{region 'Components'}
// Pumps/Engines 
  fbLowPressurePump:                              FB_PUMP_WITH_BYPASS( itfOpMode:= PrgOrg.fbOpMode, 
                                                                       itfEventLogger:= PrgOrg.fbEventLogger,
                                                                       itfOn:= fbEngine_LowPressurePump_Start,
                                                                       itfBypassValve:= fbValve_LowPressureCircuit_Enable);
  fbOilCooler:                                    FB_PUMP(itfOpMode:= PrgOrg.fbOpMode,  
                                                          itfEventLogger:= PrgOrg.fbEventLogger,
                                                          itfOn:= fbEngine_OilCooler_Start);
  fbBypassPump:                                   FB_PUMP(itfOpMode:= PrgOrg.fbOpMode, 
                                                          itfEventLogger:= PrgOrg.fbEventLogger,
                                                          itfOn:= fbEngine_BypassPump_Start);
  fbCounterCyl1Pump:                              FB_PUMP_WITH_BYPASS( itfOpMode:= PrgOrg.fbOpMode, 
                                                                       itfEventLogger:= PrgOrg.fbEventLogger,
                                                                       itfOn:= fbEngine_CounterCyl1Pump_Start,
                                                                       itfBypassValve:= fbValve_CounterCyl1_Bypass);
  fbCounterCyl2Pump:                              FB_PUMP_WITH_BYPASS( itfOpMode:= PrgOrg.fbOpMode, 
                                                                       itfEventLogger:= PrgOrg.fbEventLogger,
                                                                       itfOn:= fbEngine_CounterCyl2Pump_Start,
                                                                       itfBypassValve:= fbValve_CounterCyl2_Bypass);
  fbCounterCyl3Pump:                              FB_PUMP_WITH_BYPASS( itfOpMode:= PrgOrg.fbOpMode, 
                                                                       itfEventLogger:= PrgOrg.fbEventLogger,
                                                                       itfOn:= fbEngine_CounterCyl3Pump_Start,
                                                                       itfBypassValve:= fbValve_CounterCyl3_Bypass);
  fbCounterCyl4Pump:                              FB_PUMP_WITH_BYPASS( itfOpMode:= PrgOrg.fbOpMode,  
                                                                       itfEventLogger:= PrgOrg.fbEventLogger,
                                                                       itfOn:= fbEngine_CounterCyl4Pump_Start,
                                                                       itfBypassValve:= fbValve_CounterCyl4_Bypass);
  fbTestCyl1Pump:                                 FB_PUMP(itfOpMode:= PrgOrg.fbOpMode, 
                                                          itfEventLogger:= PrgOrg.fbEventLogger,
                                                          itfOn:= fbEngine_TestCyl1Pump_Start);
  fbTestCyl2Pump:                                 FB_PUMP(itfOpMode:= PrgOrg.fbOpMode, 
                                                          itfEventLogger:= PrgOrg.fbEventLogger,
                                                          itfOn:= fbEngine_TestCyl2Pump_Start);
  fbTestCyl3Pump:                                 FB_PUMP(itfOpMode:= PrgOrg.fbOpMode, 
                                                          itfEventLogger:= PrgOrg.fbEventLogger, 
                                                          itfOn:= fbEngine_TestCyl3Pump_Start);
  fbTestCyl4Pump:                                 FB_PUMP(itfOpMode:= PrgOrg.fbOpMode, 
                                                          itfEventLogger:= PrgOrg.fbEventLogger, 
                                                          itfOn:= fbEngine_TestCyl4Pump_Start);
      
// Valves
  fbShutOffValve_LowPressure:                     FB_SHUTOFF_VALVE( itfOpMode:= PrgOrg.fbOpMode,  
                                                                    itfEventLogger:= PrgOrg.fbEventLogger,
	                                                                  itfOpen:= fbShutOffValve_Open, 
	                                                                  itfClose:= fbShutOffValve_Close,
                                                                    itfSensorOpened:= fbShutOffValve_Opened,
                                                                    itfSensorClosed:= fbShutOffValve_Closed,
                                                                    bNC:= TRUE);
  fbValve_LowPressureCircuit_Enable:              FB_VALVE_X_2( itfOpMode:= PrgOrg.fbOpMode, 
                                                                itfEventLogger:= PrgOrg.fbEventLogger,
	                                                              itfSwitchToWP:= fbValve42_LowPressureCircuit_Enable);
  fbValve_CounterCyl1_LowPressureCircuit_Add:     FB_VALVE_X_2( itfOpMode:= PrgOrg.fbOpMode, 
                                                                itfEventLogger:= PrgOrg.fbEventLogger,
	                                                              itfSwitchToWP:= fbValve42_CounterCyl1_LowPressureCircuit_Add);
  fbValve_CounterCyl2_LowPressureCircuit_Add:     FB_VALVE_X_2( itfOpMode:= PrgOrg.fbOpMode, 
                                                                itfEventLogger:= PrgOrg.fbEventLogger,
	                                                              itfSwitchToWP:= fbValve42_CounterCyl2_LowPressureCircuit_Add);
  fbValve_CounterCyl3_LowPressureCircuit_Add:     FB_VALVE_X_2( itfOpMode:= PrgOrg.fbOpMode, 
                                                                itfEventLogger:= PrgOrg.fbEventLogger,
	                                                              itfSwitchToWP:= fbValve42_CounterCyl3_LowPressureCircuit_Add);
  fbValve_CounterCyl4_LowPressureCircuit_Add:     FB_VALVE_X_2( itfOpMode:= PrgOrg.fbOpMode,  
                                                                itfEventLogger:= PrgOrg.fbEventLogger,
	                                                              itfSwitchToWP:= fbValve42_CounterCyl4_LowPressureCircuit_Add);
  fbValve_CounterCyl1:                            FB_VALVE_X_3( itfOpMode:= PrgOrg.fbOpMode, 
                                                                itfEventLogger:= PrgOrg.fbEventLogger,
	                                                              itfSwitchToWP1:= fbValve43_CounterCyl1_Extend, 
	                                                              itfSwitchToWP2:= fbValve43_CounterCyl1_Retract);
  fbValve_CounterCyl2:                            FB_VALVE_X_3( itfOpMode:= PrgOrg.fbOpMode, 
                                                                itfEventLogger:= PrgOrg.fbEventLogger,
	                                                              itfSwitchToWP1:= fbValve43_CounterCyl2_Extend, 
	                                                              itfSwitchToWP2:= fbValve43_CounterCyl2_Retract);
  fbValve_CounterCyl3:                            FB_VALVE_X_3( itfOpMode:= PrgOrg.fbOpMode, 
                                                                itfEventLogger:= PrgOrg.fbEventLogger,
	                                                              itfSwitchToWP1:= fbValve43_CounterCyl3_Extend, 
	                                                              itfSwitchToWP2:= fbValve43_CounterCyl3_Retract);
  fbValve_CounterCyl4:                            FB_VALVE_X_3( itfOpMode:= PrgOrg.fbOpMode, 
                                                                itfEventLogger:= PrgOrg.fbEventLogger,
	                                                              itfSwitchToWP1:= fbValve43_CounterCyl4_Extend, 
	                                                              itfSwitchToWP2:= fbValve43_CounterCyl4_Retract);
  fbValve_CounterCyl1JogAutoMode:                 FB_VALVE_X_2( itfOpMode:= PrgOrg.fbOpMode, 
                                                                itfEventLogger:= PrgOrg.fbEventLogger,
	                                                              itfSwitchToWP:= fbValve22_CounterCyl1_JogMode_Off);
  fbValve_CounterCyl2JogAutoMode:                 FB_VALVE_X_2( itfOpMode:= PrgOrg.fbOpMode, 
                                                                itfEventLogger:= PrgOrg.fbEventLogger,
	                                                              itfSwitchToWP:= fbValve22_CounterCyl2_JogMode_Off);
  fbValve_CounterCyl3JogAutoMode:                 FB_VALVE_X_2( itfOpMode:= PrgOrg.fbOpMode, 
                                                                itfEventLogger:= PrgOrg.fbEventLogger,
	                                                              itfSwitchToWP:= fbValve22_CounterCyl3_JogMode_Off);
  fbValve_CounterCyl4JogAutoMode:                 FB_VALVE_X_2( itfOpMode:= PrgOrg.fbOpMode,  
                                                                itfEventLogger:= PrgOrg.fbEventLogger,
	                                                              itfSwitchToWP:= fbValve22_CounterCyl4_JogMode_Off);
  fbValve_CounterCyl1_SinkBlock:                  FB_VALVE_X_2( itfOpMode:= PrgOrg.fbOpMode,  
                                                                itfEventLogger:= PrgOrg.fbEventLogger,
	                                                              itfSwitchToWP:= fbValve22_CounterCyl1_SinkBlock_Open);
  fbValve_CounterCyl2_SinkBlock:                  FB_VALVE_X_2( itfOpMode:= PrgOrg.fbOpMode,  
                                                                itfEventLogger:= PrgOrg.fbEventLogger,
	                                                              itfSwitchToWP:= fbValve22_CounterCyl2_SinkBlock_Open);
  fbValve_CounterCyl3_SinkBlock:                  FB_VALVE_X_2( itfOpMode:= PrgOrg.fbOpMode,  
                                                                itfEventLogger:= PrgOrg.fbEventLogger,
	                                                              itfSwitchToWP:= fbValve22_CounterCyl3_SinkBlock_Open);
  fbValve_CounterCyl4_SinkBlock:                  FB_VALVE_X_2( itfOpMode:= PrgOrg.fbOpMode,  
                                                                itfEventLogger:= PrgOrg.fbEventLogger,
	                                                              itfSwitchToWP:= fbValve22_CounterCyl4_SinkBlock_Open);
  fbValve_CounterCyl1_WorkPressure:               FB_PRV_PROP(itfOpMode:= PrgOrg.fbOpMode, 
                                                              itfEventLogger:= PrgOrg.fbEventLogger,
                                                              rMaxLimitInBar:= 275.0);
  fbValve_CounterCyl2_WorkPressure:               FB_PRV_PROP(itfOpMode:= PrgOrg.fbOpMode, 
                                                              itfEventLogger:= PrgOrg.fbEventLogger,
                                                              rMaxLimitInBar:= 275.0);
  fbValve_CounterCyl3_WorkPressure:               FB_PRV_PROP(itfOpMode:= PrgOrg.fbOpMode, 
                                                              itfEventLogger:= PrgOrg.fbEventLogger,
                                                              rMaxLimitInBar:= 275.0);
  fbValve_CounterCyl4_WorkPressure:               FB_PRV_PROP(itfOpMode:= PrgOrg.fbOpMode, 
                                                              itfEventLogger:= PrgOrg.fbEventLogger,
                                                              rMaxLimitInBar:= 275.0);
  fbValve_CounterCyl1_Bypass:                     FB_VALVE_X_2( itfOpMode:= PrgOrg.fbOpMode, 
                                                                itfEventLogger:= PrgOrg.fbEventLogger,
	                                                              itfSwitchToWP:= fbValve42_CounterCyl1_Bypass_Add);
  fbValve_CounterCyl2_Bypass:                     FB_VALVE_X_2( itfOpMode:= PrgOrg.fbOpMode, 
                                                                itfEventLogger:= PrgOrg.fbEventLogger, 
	                                                              itfSwitchToWP:= fbValve42_CounterCyl2_Bypass_Add);
  fbValve_CounterCyl3_Bypass:                     FB_VALVE_X_2( itfOpMode:= PrgOrg.fbOpMode,  
                                                                itfEventLogger:= PrgOrg.fbEventLogger,
	                                                              itfSwitchToWP:= fbValve42_CounterCyl3_Bypass_Add);
  fbValve_CounterCyl4_Bypass:                     FB_VALVE_X_2( itfOpMode:= PrgOrg.fbOpMode, 
                                                                itfEventLogger:= PrgOrg.fbEventLogger,
	                                                              itfSwitchToWP:= fbValve42_CounterCyl4_Bypass_Add);
  fbValve_TestCyl1:                               FB_VALVE_X_3_PROP(itfOpMode:= PrgOrg.fbOpMode, 
                                                                    itfEventLogger:= PrgOrg.fbEventLogger);
  fbValve_TestCyl2:                               FB_VALVE_X_3_PROP(itfOpMode:= PrgOrg.fbOpMode, 
                                                                    itfEventLogger:= PrgOrg.fbEventLogger);
  fbValve_TestCyl3:                               FB_VALVE_X_3_PROP(itfOpMode:= PrgOrg.fbOpMode, 
                                                                    itfEventLogger:= PrgOrg.fbEventLogger);
  fbValve_TestCyl4:                               FB_VALVE_X_3_PROP(itfOpMode:= PrgOrg.fbOpMode, 
                                                                    itfEventLogger:= PrgOrg.fbEventLogger);
  fbValve_TestCyl1_A_Unlock:                      FB_VALVE_X_2( itfOpMode:= PrgOrg.fbOpMode, 
                                                                itfEventLogger:= PrgOrg.fbEventLogger,
	                                                              itfSwitchToWP:= fbValve22_TestCyl1_A_Open);
  fbValve_TestCyl1_B_Unlock:                      FB_VALVE_X_2( itfOpMode:= PrgOrg.fbOpMode, 
                                                                itfEventLogger:= PrgOrg.fbEventLogger, 
	                                                              itfSwitchToWP:= fbValve22_TestCyl1_B_Open);
  fbValve_TestCyl2_A_Unlock:                      FB_VALVE_X_2( itfOpMode:= PrgOrg.fbOpMode,   
                                                                itfEventLogger:= PrgOrg.fbEventLogger, 
	                                                              itfSwitchToWP:= fbValve22_TestCyl2_A_Open);
  fbValve_TestCyl2_B_Unlock:                      FB_VALVE_X_2( itfOpMode:= PrgOrg.fbOpMode, 
                                                                itfEventLogger:= PrgOrg.fbEventLogger,  
	                                                              itfSwitchToWP:= fbValve22_TestCyl2_B_Open);
  fbValve_TestCyl3_A_Unlock:                      FB_VALVE_X_2( itfOpMode:= PrgOrg.fbOpMode,  
                                                                itfEventLogger:= PrgOrg.fbEventLogger,
	                                                              itfSwitchToWP:= fbValve22_TestCyl3_A_Open);
  fbValve_TestCyl3_B_Unlock:                      FB_VALVE_X_2( itfOpMode:= PrgOrg.fbOpMode,  
                                                                itfEventLogger:= PrgOrg.fbEventLogger,
	                                                              itfSwitchToWP:= fbValve22_TestCyl3_B_Open);
  fbValve_TestCyl4_A_Unlock:                      FB_VALVE_X_2( itfOpMode:= PrgOrg.fbOpMode, 
                                                                itfEventLogger:= PrgOrg.fbEventLogger,
	                                                              itfSwitchToWP:= fbValve22_TestCyl4_A_Open);
  fbValve_TestCyl4_B_Unlock:                      FB_VALVE_X_2( itfOpMode:= PrgOrg.fbOpMode, 
                                                                itfEventLogger:= PrgOrg.fbEventLogger,
	                                                              itfSwitchToWP:= fbValve22_TestCyl4_B_Open);
  fbValve_TestCyl1_WorkPressure:                  FB_PRV_PROP(itfOpMode:= PrgOrg.fbOpMode, 
                                                              itfEventLogger:= PrgOrg.fbEventLogger,
                                                              rMaxLimitInBar:= 275.0);
  fbValve_TestCyl2_WorkPressure:                  FB_PRV_PROP(itfOpMode:= PrgOrg.fbOpMode, 
                                                              itfEventLogger:= PrgOrg.fbEventLogger,
                                                              rMaxLimitInBar:= 275.0);
  fbValve_TestCyl3_WorkPressure:                  FB_PRV_PROP(itfOpMode:= PrgOrg.fbOpMode, 
                                                              itfEventLogger:= PrgOrg.fbEventLogger,
                                                              rMaxLimitInBar:= 275.0);
  fbValve_TestCyl4_WorkPressure:                  FB_PRV_PROP(itfOpMode:= PrgOrg.fbOpMode, 
                                                              itfEventLogger:= PrgOrg.fbEventLogger,
                                                              rMaxLimitInBar:= 275.0);
  fbValve_TestCyl1_LowPressure:                   FB_PRV_PROP(itfOpMode:= PrgOrg.fbOpMode, 
                                                              itfEventLogger:= PrgOrg.fbEventLogger,
                                                              rMaxLimitInBar:= 25.0);
  fbValve_Pump4_Add:                              FB_VALVE_X_2( itfOpMode:= PrgOrg.fbOpMode, 
                                                                itfEventLogger:= PrgOrg.fbEventLogger,
	                                                              itfSwitchToWP:= fbValve22_Pump4_Add);
  fbValve_Pump3_Add:                              FB_VALVE_X_2( itfOpMode:= PrgOrg.fbOpMode,  
                                                                itfEventLogger:= PrgOrg.fbEventLogger,
	                                                              itfSwitchToWP:= fbValve22_Pump3_Add);
  fbValve_Pump2_Add:                              FB_VALVE_X_2( itfOpMode:= PrgOrg.fbOpMode,  
                                                                itfEventLogger:= PrgOrg.fbEventLogger,
	                                                              itfSwitchToWP:= fbValve22_Pump2_Add);
  fbValve_PressureReservoir_A_Add:                FB_VALVE_X_2( itfOpMode:= PrgOrg.fbOpMode, 
                                                                itfEventLogger:= PrgOrg.fbEventLogger, 
	                                                              itfSwitchToWP:= fbValve22_PressureReservoir_A_Add);
  fbValve_PressureReservoir_B_Add:                FB_VALVE_X_2( itfOpMode:= PrgOrg.fbOpMode, 
                                                                itfEventLogger:= PrgOrg.fbEventLogger,
	                                                              itfSwitchToWP:= fbValve22_PressureReservoir_B_Add);
  fbValve_SensorBreakPressure_A_Add:              FB_VALVE_X_2( itfOpMode:= PrgOrg.fbOpMode, 
                                                                itfEventLogger:= PrgOrg.fbEventLogger,
	                                                              itfSwitchToWP:= fbValve32_SensorBreakPressure_A_Add);
  fbValve_SensorBreakPressure_B_Add:              FB_VALVE_X_2( itfOpMode:= PrgOrg.fbOpMode, 
                                                                itfEventLogger:= PrgOrg.fbEventLogger,
	                                                              itfSwitchToWP:= fbValve32_SensorBreakPressure_B_Add);
                                                  
// Cylinders                                      
  fbCounterCyl1:                                  FB_CYLINDER_DA_COUNTER( itfOpMode:= PrgOrg.fbOpMode, 
                                                                          itfEventLogger:= PrgOrg.fbEventLogger,
                                                                          itfOpModeVisu:= PrgVisu.fbVisuOPMode,
                                                                          itfValve_CylCtrl:= fbValve_CounterCyl1,
                                                                          itfValve_Bypass:= fbValve_CounterCyl1_Bypass,
                                                                          itfValve_AutomaticEnable:= fbValve_CounterCyl1JogAutoMode,
                                                                          itfValve_SinkBlock:= fbValve_CounterCyl1_SinkBlock,
                                                                          itfValve_LowPressureCircuitAdd:= fbValve_CounterCyl1_LowPressureCircuit_Add,
                                                                          itfValve_PressureLimit:= fbValve_CounterCyl1_WorkPressure,
                                                                          itfJogBtnPos_Pressed:= fbJogBtnPos_Pressed,
                                                                          itfJogBtnNeg_Pressed:= fbJogBtnNeg_Pressed,
	                                                                        lrPistonSurfaceA:= 1963.495, 
	                                                                        lrPistonSurfaceB:= 962.112, 
	                                                                        rEndPosTol:= 1,
                                                                          rPumpVolumeFlow:= 4.0,
                                                                          rPumpEfficiencyFactor:= 0.85);
  fbCounterCyl2:                                  FB_CYLINDER_DA_COUNTER( itfOpMode:= PrgOrg.fbOpMode, 
                                                                          itfEventLogger:= PrgOrg.fbEventLogger,
                                                                          itfOpModeVisu:= PrgVisu.fbVisuOPMode,
                                                                          itfValve_CylCtrl:= fbValve_CounterCyl2,
                                                                          itfValve_Bypass:= fbValve_CounterCyl2_Bypass,
                                                                          itfValve_AutomaticEnable:= fbValve_CounterCyl2JogAutoMode,
                                                                          itfValve_SinkBlock:= fbValve_CounterCyl2_SinkBlock,
                                                                          itfValve_LowPressureCircuitAdd:= fbValve_CounterCyl2_LowPressureCircuit_Add,
                                                                          itfValve_PressureLimit:= fbValve_CounterCyl2_WorkPressure,
                                                                          itfJogBtnPos_Pressed:= fbJogBtnPos_Pressed,
                                                                          itfJogBtnNeg_Pressed:= fbJogBtnNeg_Pressed,
	                                                                        lrPistonSurfaceA:= 1963.495, 
	                                                                        lrPistonSurfaceB:= 962.112, 
	                                                                        rEndPosTol:= 1,
                                                                          rPumpVolumeFlow:= 4.0,
                                                                          rPumpEfficiencyFactor:= 0.85);
  fbCounterCyl3:                                  FB_CYLINDER_DA_COUNTER( itfOpMode:= PrgOrg.fbOpMode, 
                                                                          itfEventLogger:= PrgOrg.fbEventLogger,
                                                                          itfOpModeVisu:= PrgVisu.fbVisuOPMode,
                                                                          itfValve_CylCtrl:= fbValve_CounterCyl3,
                                                                          itfValve_Bypass:= fbValve_CounterCyl3_Bypass,
                                                                          itfValve_AutomaticEnable:= fbValve_CounterCyl3JogAutoMode,
                                                                          itfValve_SinkBlock:= fbValve_CounterCyl3_SinkBlock,
                                                                          itfValve_LowPressureCircuitAdd:= fbValve_CounterCyl3_LowPressureCircuit_Add,
                                                                          itfValve_PressureLimit:= fbValve_CounterCyl3_WorkPressure,
                                                                          itfJogBtnPos_Pressed:= fbJogBtnPos_Pressed,
                                                                          itfJogBtnNeg_Pressed:= fbJogBtnNeg_Pressed,
	                                                                        lrPistonSurfaceA:= 1963.495, 
	                                                                        lrPistonSurfaceB:= 962.112, 
	                                                                        rEndPosTol:= 1,
                                                                          rPumpVolumeFlow:= 4.0,
                                                                          rPumpEfficiencyFactor:= 0.85);
  fbCounterCyl4:                                  FB_CYLINDER_DA_COUNTER( itfOpMode:= PrgOrg.fbOpMode, 
                                                                          itfEventLogger:= PrgOrg.fbEventLogger,
                                                                          itfOpModeVisu:= PrgVisu.fbVisuOPMode,
                                                                          itfValve_CylCtrl:= fbValve_CounterCyl4,
                                                                          itfValve_Bypass:= fbValve_CounterCyl4_Bypass,
                                                                          itfValve_AutomaticEnable:= fbValve_CounterCyl4JogAutoMode,
                                                                          itfValve_SinkBlock:= fbValve_CounterCyl4_SinkBlock,
                                                                          itfValve_LowPressureCircuitAdd:= fbValve_CounterCyl4_LowPressureCircuit_Add,
                                                                          itfValve_PressureLimit:= fbValve_CounterCyl4_WorkPressure,  
                                                                          itfJogBtnPos_Pressed:= fbJogBtnPos_Pressed,
                                                                          itfJogBtnNeg_Pressed:= fbJogBtnNeg_Pressed,
	                                                                        lrPistonSurfaceA:= 1963.495, 
	                                                                        lrPistonSurfaceB:= 962.112, 
	                                                                        rEndPosTol:= 1,
                                                                          rPumpVolumeFlow:= 4.0,
                                                                          rPumpEfficiencyFactor:= 0.85);
  fbTestCyl1:                                     FB_CYLINDER_DA_TESTDEV1(itfOpMode:= PrgOrg.fbOpMode, 
                                                                          itfEventLogger:= PrgOrg.fbEventLogger, 
                                                                          itfOpModeVisu:= PrgVisu.fbVisuOPMode,
	                                                                        itfValve_CylCtrl:= fbValve_TestCyl1, 
	                                                                        itfValve_LockA:= fbValve_TestCyl1_A_Unlock, 
	                                                                        itfValve_LockB:= fbValve_TestCyl1_B_Unlock, 
	                                                                        itfValve_AddPump2:= fbValve_Pump2_Add, 
	                                                                        itfValve_AddPump3:= fbValve_Pump3_Add, 
	                                                                        itfValve_AddPump4:= fbValve_Pump4_Add, 
	                                                                        itfValve_PressureReservoirAAdd:= fbValve_PressureReservoir_A_Add, 
	                                                                        itfValve_PressureReservoirBAdd:= fbValve_PressureReservoir_B_Add, 
	                                                                        itfValve_SensorBreakPressureAAdd:= fbValve_SensorBreakPressure_A_Add, 
	                                                                        itfValve_SensorBreakPressureBAdd:= fbValve_SensorBreakPressure_B_Add, 
	                                                                        fbShutOffValve_LowPressure:= fbShutOffValve_LowPressure, 
	                                                                        itfValve_PressureLimit:= fbValve_TestCyl1_WorkPressure, 
	                                                                        itfValve_LowPressureLimit:= fbValve_TestCyl1_LowPressure,
                                                                          itfPumpMain:= fbTestCyl1Pump,
                                                                          itfPump2:= fbTestCyl2Pump, 
                                                                          itfPump3:= fbTestCyl3Pump, 
                                                                          itfPump4:= fbTestCyl4Pump, 
	                                                                        rEndPosTol:= 1,
                                                                          rPumpVolumeFlow:= 3.0,
                                                                          rPumpEfficiencyFactor:= 0.85);
  fbTestCyl2:                                     FB_CYLINDER_DA_TESTDEV2_4(itfOpMode:= PrgOrg.fbOpMode, 
                                                                            itfEventLogger:= PrgOrg.fbEventLogger,
                                                                            itfOpModeVisu:= PrgVisu.fbVisuOPMode,
	                                                                          itfValve_CylCtrl:= fbValve_TestCyl2, 
	                                                                          itfValve_LockA:= fbValve_TestCyl2_A_Unlock, 
	                                                                          itfValve_LockB:= fbValve_TestCyl2_B_Unlock, 
	                                                                          itfValve_PressureLimit:= fbValve_TestCyl2_WorkPressure,
	                                                                          rEndPosTol:= 1,
                                                                            rPumpVolumeFlow:= 3.0,
                                                                            rPumpEfficiencyFactor:= 0.85);
  fbTestCyl3:                                     FB_CYLINDER_DA_TESTDEV2_4(itfOpMode:= PrgOrg.fbOpMode,  
                                                                            itfEventLogger:= PrgOrg.fbEventLogger,
                                                                            itfOpModeVisu:= PrgVisu.fbVisuOPMode,
	                                                                          itfValve_CylCtrl:= fbValve_TestCyl3, 
	                                                                          itfValve_LockA:= fbValve_TestCyl3_A_Unlock, 
	                                                                          itfValve_LockB:= fbValve_TestCyl3_B_Unlock, 
	                                                                          itfValve_PressureLimit:= fbValve_TestCyl3_WorkPressure, 
	                                                                          rEndPosTol:= 1,
                                                                            rPumpVolumeFlow:= 3.0,
                                                                            rPumpEfficiencyFactor:= 0.85);
  fbTestCyl4:                                     FB_CYLINDER_DA_TESTDEV2_4(itfOpMode:= PrgOrg.fbOpMode, 
                                                                            itfEventLogger:= PrgOrg.fbEventLogger,
                                                                            itfOpModeVisu:= PrgVisu.fbVisuOPMode,
	                                                                          itfValve_CylCtrl:= fbValve_TestCyl4, 
	                                                                          itfValve_LockA:= fbValve_TestCyl4_A_Unlock, 
	                                                                          itfValve_LockB:= fbValve_TestCyl4_B_Unlock, 
	                                                                          itfValve_PressureLimit:= fbValve_TestCyl4_WorkPressure,
	                                                                          rEndPosTol:= 1,
                                                                            rPumpVolumeFlow:= 3.0,
                                                                            rPumpEfficiencyFactor:= 0.85);
{endregion}
   
{region 'Main process'}
  fbNest1:                                        FB_SEQ_PROCESS_NEST1( itfOpMode:= PrgOrg.fbOpMode, 
                                                                        itfEventLogger:= PrgOrg.fbEventLogger,
                                                                        itfTimer:= fbTimerNest1, 
	                                                                      itfCounterCyl:= fbCounterCyl1, 
	                                                                      itfTestCyl:= fbTestCyl1, 
	                                                                      itfCounterCylPump:= fbCounterCyl1Pump, 
	                                                                      itfTestCylPump:= fbTestCyl1Pump,
                                                                        itfPump2Pressure:= fbValve_TestCyl2_WorkPressure,
                                                                        itfPump3Pressure:= fbValve_TestCyl3_WorkPressure,
                                                                        itfPump4Pressure:= fbValve_TestCyl4_WorkPressure);
  fbNest2:                                        FB_SEQ_PROCESS_NEST2_4( itfOpMode:= PrgOrg.fbOpMode, 
                                                                          itfEventLogger:= PrgOrg.fbEventLogger,
                                                                          itfTimer:= fbTimerNest2, 
	                                                                        itfCounterCyl:= fbCounterCyl2, 
	                                                                        itfTestCyl:= fbTestCyl2, 
	                                                                        itfCounterCylPump:= fbCounterCyl2Pump, 
	                                                                        itfTestCylPump:= fbTestCyl2Pump);
  fbNest3:                                        FB_SEQ_PROCESS_NEST2_4( itfOpMode:= PrgOrg.fbOpMode,  
                                                                          itfEventLogger:= PrgOrg.fbEventLogger,
                                                                          itfTimer:= fbTimerNest3,
	                                                                        itfCounterCyl:= fbCounterCyl3, 
	                                                                        itfTestCyl:= fbTestCyl3, 
	                                                                        itfCounterCylPump:= fbCounterCyl3Pump, 
	                                                                        itfTestCylPump:= fbTestCyl3Pump);
  fbNest4:                                        FB_SEQ_PROCESS_NEST2_4( itfOpMode:= PrgOrg.fbOpMode,  
                                                                          itfEventLogger:= PrgOrg.fbEventLogger,
                                                                          itfTimer:= fbTimerNest4,
	                                                                        itfCounterCyl:= fbCounterCyl4, 
	                                                                        itfTestCyl:= fbTestCyl4, 
	                                                                        itfCounterCylPump:= fbCounterCyl4Pump, 
	                                                                        itfTestCylPump:= fbTestCyl4Pump);
  fbMainProcess:                                  FB_PROCESS_MAIN(itfOpMode:= PrgOrg.fbOpMode, 
                                                                  itfEventLogger:= PrgOrg.fbEventLogger, 
                                                                  itfTimerNest1:= fbTimerNest1,
                                                                  itfTimerNest2:= fbTimerNest2,
                                                                  itfTimerNest3:= fbTimerNest3,
                                                                  itfTimerNest4:= fbTimerNest4,
	                                                                itfNest1:= fbNest1, 
	                                                                itfNest2:= fbNest2, 
	                                                                itfNest3:= fbNest3, 
	                                                                itfNest4:= fbNest4, 
	                                                                itfLowPressurePump:= fbLowPressurePump, 
	                                                                itfOilCooler:= fbOilCooler, 
	                                                                itfBypassPump:= fbBypassPump,
                                                                  itfLevelSwitch_AggregateTank1_Out1:= fbLevelSwitch_AggregateTank1_Out1,
                                                                  itfLevelSwitch_AggregateTank1_Out2:= fbLevelSwitch_AggregateTank1_Out2,
                                                                  itfTemperatureSwitch_AggregateTank1_Out1:= fbTemperatureSwitch_AggregateTank1_Out1,
                                                                  itfTemperatureSwitch_AggregateTank1_Out2:= fbTemperatureSwitch_AggregateTank1_Out2,
                                                                  itfLevelSwitch_AggregateTank2_Out1:= fbLevelSwitch_AggregateTank2_Out1,
                                                                  itfLevelSwitch_AggregateTank2_Out2:= fbLevelSwitch_AggregateTank2_Out2,
                                                                  itfLevelSwitch_AggregateTank2_Out3:= fbLevelSwitch_AggregateTank2_Out3,
                                                                  itfSwitch_AggregateFilter_Dirty:= fbSwitch_AggregateFilter_Dirty);
{endregion}
   
{region 'Recipe'}
  stRecipeParams:                                 ST_RECIPE_PARAMS;
{endregion}
END_VAR
VAR
  rMaxSpeedInMmPerSHP:                            REAL;
  rMaxSpeedInMmPerSWP:                            REAL;
END_VAR

VAR PERSISTENT
  stSettings:                                     ST_SETTINGS;
  sTestCyl1SNo:                                   STRING := '';
  sTestCyl2SNo:                                   STRING := '';
  sTestCyl3SNo:                                   STRING := '';
  sTestCyl4SNo:                                   STRING := '';
END_VAR

(* Actions *)
A_000_FBs();
A_010_InputToBNC();
A_020_SetObjectPath();
A_030_OilCooler();
A_040_MachineLight();
A_100_Control();

ACTION A_000_FBs:
(* FBs *)
// General
fbTimerNest1();
fbTimerNest2();
fbTimerNest3();
fbTimerNest4();
rPressureConverted_TestCyl1 := TO_REAL(iPressureSensor_TestCyl1) * 0.025;
rPressureConverted_TestCyl1_A := TO_REAL(iPressureSensor_TestCyl1_A) * 0.025;
rPressureConverted_TestCyl1_B := TO_REAL(iPressureSensor_TestCyl1_B) * 0.025;
rPressureConverted_CounterCyl1 := TO_REAL(iPressureSensor_CounterCyl1) * 0.025;
rPressureConverted_LowPressure := TO_REAL(iPressureSensor_LowPressure) * 0.001;
rPressureConverted_TestCyl1_BreakPressure_A := TO_REAL(iPressureSensor_TestCyl1_BreakPressure_A) * 0.001;
rPressureConverted_TestCyl1_BreakPressure_B := TO_REAL(iPressureSensor_TestCyl1_BreakPressure_B) * 0.001;
rPressureConverted_TestCyl1_PressureReservoir := TO_REAL(iPressureSensor_TestCyl1_PressureReservoir) * 0.025;
rPressureConverted_TestCyl2 := TO_REAL(iPressureSensor_TestCyl2) * 0.025;
rPressureConverted_TestCyl2_A := TO_REAL(iPressureSensor_TestCyl2_A) * 0.025;
rPressureConverted_TestCyl2_B := TO_REAL(iPressureSensor_TestCyl2_B) * 0.025;
rPressureConverted_CounterCyl2 := TO_REAL(iPressureSensor_CounterCyl2) * 0.025;
rPressureConverted_TestCyl3 := TO_REAL(iPressureSensor_TestCyl3) * 0.025;
rPressureConverted_TestCyl3_A := TO_REAL(iPressureSensor_TestCyl3_A) * 0.025;
rPressureConverted_TestCyl3_B := TO_REAL(iPressureSensor_TestCyl3_B) * 0.025;
rPressureConverted_CounterCyl3 := TO_REAL(iPressureSensor_CounterCyl3) * 0.025;
rPressureConverted_TestCyl4 := TO_REAL(iPressureSensor_TestCyl4) * 0.025;
rPressureConverted_TestCyl4_A := TO_REAL(iPressureSensor_TestCyl4_A) * 0.025;
rPressureConverted_TestCyl4_B := TO_REAL(iPressureSensor_TestCyl4_B) * 0.025;
rPressureConverted_CounterCyl4 := TO_REAL(iPressureSensor_CounterCyl4) * 0.025;


// Pmps/Engines
fbLowPressurePump();
fbOilCooler();
fbBypassPump();
fbCounterCyl1Pump();
fbCounterCyl2Pump();
fbCounterCyl3Pump();
fbCounterCyl4Pump();
fbTestCyl1Pump();
fbTestCyl2Pump();
fbTestCyl3Pump();
fbTestCyl4Pump();
fbShutOffValve_LowPressure();

// Valves
fbValve_LowPressureCircuit_Enable();
fbValve_CounterCyl1_LowPressureCircuit_Add();
fbValve_CounterCyl2_LowPressureCircuit_Add();
fbValve_CounterCyl3_LowPressureCircuit_Add();
fbValve_CounterCyl4_LowPressureCircuit_Add();
fbValve_CounterCyl1();
fbValve_CounterCyl2();
fbValve_CounterCyl3();
fbValve_CounterCyl4();
fbValve_CounterCyl1JogAutoMode();
fbValve_CounterCyl2JogAutoMode();
fbValve_CounterCyl3JogAutoMode();
fbValve_CounterCyl4JogAutoMode();
fbValve_CounterCyl1_SinkBlock();
fbValve_CounterCyl2_SinkBlock();
fbValve_CounterCyl3_SinkBlock();
fbValve_CounterCyl4_SinkBlock();
fbValve_CounterCyl1_WorkPressure(iTargetVal=> iCounterCyl1_Pressure);
fbValve_CounterCyl2_WorkPressure(iTargetVal=> iCounterCyl2_Pressure);
fbValve_CounterCyl3_WorkPressure(iTargetVal=> iCounterCyl3_Pressure);
fbValve_CounterCyl4_WorkPressure(iTargetVal=> iCounterCyl4_Pressure);
fbValve_CounterCyl1_Bypass();
fbValve_CounterCyl2_Bypass();
fbValve_CounterCyl3_Bypass();
fbValve_CounterCyl4_Bypass();
fbValve_TestCyl1(iAnalogSwitch=> iValve43_TestCyl1);
fbValve_TestCyl2(iAnalogSwitch=> iValve43_TestCyl2);
fbValve_TestCyl3(iAnalogSwitch=> iValve43_TestCyl3);
fbValve_TestCyl4(iAnalogSwitch=> iValve43_TestCyl4);
fbValve_TestCyl1_A_Unlock();
fbValve_TestCyl1_B_Unlock();
fbValve_TestCyl2_A_Unlock();
fbValve_TestCyl2_B_Unlock();
fbValve_TestCyl3_A_Unlock();
fbValve_TestCyl3_B_Unlock();
fbValve_TestCyl4_A_Unlock();
fbValve_TestCyl4_B_Unlock();
fbValve_TestCyl1_WorkPressure(iTargetVal=> iTestCyl1_Pressure);
fbValve_TestCyl2_WorkPressure(iTargetVal=> iTestCyl2_Pressure);
fbValve_TestCyl3_WorkPressure(iTargetVal=> iTestCyl3_Pressure);
fbValve_TestCyl4_WorkPressure(iTargetVal=> iTestCyl4_Pressure);
fbValve_TestCyl1_LowPressure(iTargetVal=> iTestCyl1_LowPressure);
fbValve_Pump4_Add();
fbValve_Pump3_Add();
fbValve_Pump2_Add();
fbValve_PressureReservoir_A_Add();
fbValve_PressureReservoir_B_Add();
fbValve_SensorBreakPressure_A_Add();
fbValve_SensorBreakPressure_B_Add();

// Cylinders
fbCounterCyl1(rCurrentPressureInBar:= rPressureConverted_CounterCyl1, 
              bJogActive:= PrgVisu.fbVisuOPMode.P_JogCounterCyl1_Active,
              rPressureRegulationFactor:= stSettings.rPressureRegulationFactor,
              rPressureRegulationTolerance:= stSettings.rPressureRegulationTolerance);
fbCounterCyl2(rCurrentPressureInBar:= rPressureConverted_CounterCyl2, 
              bJogActive:= PrgVisu.fbVisuOPMode.P_JogCounterCyl2_Active,
              rPressureRegulationFactor:= stSettings.rPressureRegulationFactor,
              rPressureRegulationTolerance:= stSettings.rPressureRegulationTolerance);
fbCounterCyl3(rCurrentPressureInBar:= rPressureConverted_CounterCyl3, 
              bJogActive:= PrgVisu.fbVisuOPMode.P_JogCounterCyl3_Active,
              rPressureRegulationFactor:= stSettings.rPressureRegulationFactor,
              rPressureRegulationTolerance:= stSettings.rPressureRegulationTolerance);
fbCounterCyl4(rCurrentPressureInBar:= rPressureConverted_CounterCyl4, 
              bJogActive:= PrgVisu.fbVisuOPMode.P_JogCounterCyl4_Active,
              rPressureRegulationFactor:= stSettings.rPressureRegulationFactor,
              rPressureRegulationTolerance:= stSettings.rPressureRegulationTolerance);
fbTestCyl1( bDoableActing:= stRecipeParams.stRecipeCyl.bDoubleActing,
            lrCurrentPosAbs:= TO_LREAL(diTestCyl1_Distance), 
            rCurrentPressureInBar:= rPressureConverted_TestCyl1,
            rCurrentPressureInBarA:= rPressureConverted_TestCyl1_A,
            rCurrentPressureInBarB:= rPressureConverted_TestCyl1_B,
            rCurrentLowPressureInBar:= rPressureConverted_LowPressure,
            rCurrentLowPressureInBarA:= rPressureConverted_TestCyl1_BreakPressure_A,
            rCurrentLowPressureInBarB:= rPressureConverted_TestCyl1_BreakPressure_B,
            rCurrentReservoirPressureInBar:= rPressureConverted_TestCyl1_PressureReservoir,
            lrPistonSurfaceA:= stRecipeParams.stRecipeCyl.lrPistonSurfaceA,
            lrPistonSurfaceB:= stRecipeParams.stRecipeCyl.lrPistonSurfaceB,
            rSpeedRegulationFactor:= stSettings.rSpeedRegulationFactor,
            rSpeedRegulationTolerance:= stSettings.rSpeedRegulationTolerance,
            rPressureRegulationFactor:= stSettings.rPressureRegulationFactor,
            rPressureRegulationTolerance:= stSettings.rPressureRegulationTolerance);
fbTestCyl2( bDoableActing:= stRecipeParams.stRecipeCyl.bDoubleActing,
            lrCurrentPosAbs:= TO_REAL(diTestCyl2_Distance), 
            rCurrentPressureInBar:= rPressureConverted_TestCyl2,
            rCurrentPressureInBarA:= rPressureConverted_TestCyl2_A,
            rCurrentPressureInBarB:= rPressureConverted_TestCyl2_B,
            lrPistonSurfaceA:= stRecipeParams.stRecipeCyl.lrPistonSurfaceA,
            lrPistonSurfaceB:= stRecipeParams.stRecipeCyl.lrPistonSurfaceB,
            rSpeedRegulationFactor:= stSettings.rSpeedRegulationFactor,
            rSpeedRegulationTolerance:= stSettings.rSpeedRegulationTolerance,
            rPressureRegulationFactor:= stSettings.rPressureRegulationFactor,
            rPressureRegulationTolerance:= stSettings.rPressureRegulationTolerance);
fbTestCyl3( bDoableActing:= stRecipeParams.stRecipeCyl.bDoubleActing,
            lrCurrentPosAbs:= TO_REAL(diTestCyl3_Distance), 
            rCurrentPressureInBar:= rPressureConverted_TestCyl3,
            rCurrentPressureInBarA:= rPressureConverted_TestCyl3_A,
            rCurrentPressureInBarB:= rPressureConverted_TestCyl3_B,
            lrPistonSurfaceA:= stRecipeParams.stRecipeCyl.lrPistonSurfaceA,
            lrPistonSurfaceB:= stRecipeParams.stRecipeCyl.lrPistonSurfaceB,
            rSpeedRegulationFactor:= stSettings.rSpeedRegulationFactor,
            rSpeedRegulationTolerance:= stSettings.rSpeedRegulationTolerance,
            rPressureRegulationFactor:= stSettings.rPressureRegulationFactor,
            rPressureRegulationTolerance:= stSettings.rPressureRegulationTolerance);
fbTestCyl4( bDoableActing:= stRecipeParams.stRecipeCyl.bDoubleActing,
            lrCurrentPosAbs:= TO_REAL(diTestCyl4_Distance), 
            rCurrentPressureInBar:= rPressureConverted_TestCyl4,
            rCurrentPressureInBarA:= rPressureConverted_TestCyl4_A,
            rCurrentPressureInBarB:= rPressureConverted_TestCyl4_B,
            lrPistonSurfaceA:= stRecipeParams.stRecipeCyl.lrPistonSurfaceA,
            lrPistonSurfaceB:= stRecipeParams.stRecipeCyl.lrPistonSurfaceB,
            rSpeedRegulationFactor:= stSettings.rSpeedRegulationFactor,
            rSpeedRegulationTolerance:= stSettings.rSpeedRegulationTolerance,
            rPressureRegulationFactor:= stSettings.rPressureRegulationFactor,
            rPressureRegulationTolerance:= stSettings.rPressureRegulationTolerance);

// Main process
fbNest1(bDoubleActing:= stRecipeParams.stRecipeCyl.bDoubleActing,
        rMaxSpeedInMmPerSHP=> rMaxSpeedInMmPerSHP,
        rMaxSpeedInMmPerSWP=> rMaxSpeedInMmPerSWP,
        rSpeedEfficiencyFactor:= stSettings.rSpeedEfficiencyFactor,
        uiRecordDelay:= stSettings.uiRecordDelay);
fbNest2(bDoubleActing:= stRecipeParams.stRecipeCyl.bDoubleActing,
        rMaxSpeedInMmPerSHP:= rMaxSpeedInMmPerSHP,
        rMaxSpeedInMmPerSWP:= rMaxSpeedInMmPerSWP,
        rSpeedEfficiencyFactor:= stSettings.rSpeedEfficiencyFactor,
        uiRecordDelay:= stSettings.uiRecordDelay);
fbNest3(bDoubleActing:= stRecipeParams.stRecipeCyl.bDoubleActing,
        rMaxSpeedInMmPerSHP:= rMaxSpeedInMmPerSHP,
        rMaxSpeedInMmPerSWP:= rMaxSpeedInMmPerSWP,
        rSpeedEfficiencyFactor:= stSettings.rSpeedEfficiencyFactor,
        uiRecordDelay:= stSettings.uiRecordDelay);
fbNest4(bDoubleActing:= stRecipeParams.stRecipeCyl.bDoubleActing,
        rMaxSpeedInMmPerSHP:= rMaxSpeedInMmPerSHP,
        rMaxSpeedInMmPerSWP:= rMaxSpeedInMmPerSWP,
        rSpeedEfficiencyFactor:= stSettings.rSpeedEfficiencyFactor,
        uiRecordDelay:= stSettings.uiRecordDelay);
fbMainProcess();
END_ACTION

ACTION A_010_InputToBNC:
iBNCSocket_TestCyl1_A_Pressure := TO_INT(rPressureConverted_TestCyl1_A);
iBNCSocket_TestCyl1_B_Pressure := TO_INT(rPressureConverted_TestCyl1_B);
iBNCSocket_CounterCyl1_Pressure := TO_INT(rPressureConverted_CounterCyl1);
iBNCSocket_TestCyl1_Distance := TO_INT(diTestCyl1_Distance);
iBNCSocket_TestCyl1_A_BreakPressure := iPressureSensor_TestCyl1_BreakPressure_A;
iBNCSocket_TestCyl1_B_BreakPressure := iPressureSensor_TestCyl1_BreakPressure_B;
iBNCSocket_TestingCyl1_PressureReservoir := TO_INT(rPressureConverted_TestCyl1_PressureReservoir);
iBNCSocket_TestCyl2_A_Pressure := TO_INT(rPressureConverted_TestCyl2_A);
iBNCSocket_TestCyl2_B_Pressure := TO_INT(rPressureConverted_TestCyl2_B);
iBNCSocket_CounterCyl2_Pressure := TO_INT(rPressureConverted_CounterCyl2);
iBNCSocket_TestCyl2_Distance := TO_INT(diTestCyl2_Distance);
iBNCSocket_TestCyl3_A_Pressure := TO_INT(rPressureConverted_TestCyl3_A);
iBNCSocket_TestCyl3_B_Pressure := TO_INT(rPressureConverted_TestCyl3_B);
iBNCSocket_CounterCyl3_Pressure := TO_INT(rPressureConverted_CounterCyl3);
iBNCSocket_TestCyl3_Distance := TO_INT(diTestCyl3_Distance);
iBNCSocket_TestCyl4_A_Pressure := TO_INT(rPressureConverted_TestCyl4_A);
iBNCSocket_TestCyl4_B_Pressure := TO_INT(rPressureConverted_TestCyl4_B);
iBNCSocket_CounterCyl4_Pressure := TO_INT(rPressureConverted_CounterCyl4);
iBNCSocket_TestCyl4_Distance := TO_INT(diTestCyl4_Distance);
END_ACTION

ACTION A_020_SetObjectPath:
// Fbs init
fbCounterCyl1.P_FullObjectPath := 'PrgStation.fbCounterCyl1';
fbCounterCyl2.P_FullObjectPath := 'PrgStation.fbCounterCyl2';
fbCounterCyl3.P_FullObjectPath := 'PrgStation.fbCounterCyl3';
fbCounterCyl4.P_FullObjectPath := 'PrgStation.fbCounterCyl4';
fbTestCyl1.P_FullObjectPath := 'PrgStation.fbTestCyl1';
fbTestCyl2.P_FullObjectPath := 'PrgStation.fbTestCyl2';
fbTestCyl3.P_FullObjectPath := 'PrgStation.fbTestCyl3';
fbTestCyl4.P_FullObjectPath := 'PrgStation.fbTestCyl4';
END_ACTION

ACTION A_030_OilCooler:
// Bypass and oil cooler control
IF TRUE
AND NOT fbOilCooler.P_State 
THEN
  fbOilCooler.M_On();
END_IF
IF TRUE
AND NOT fbBypassPump.P_State
THEN
  fbBypassPump.M_On();
END_IF
END_ACTION

ACTION A_040_MachineLight:
IF NOT fbMachineLight.P_State AND PrgVisu.bMachineLightOn THEN
  fbMachineLight.M_Set();
END_IF

IF NOT PrgVisu.bMachineLightOn THEN
  fbMachineLight.M_Reset();
END_IF
END_ACTION

ACTION A_100_Control:
(* Control *)
iInfoOPMode := PrgOrg.fbOpMode.P_OP_MODE_STATE;
// Set ready
IF TRUE
   AND (PrgOrg.fbOpMode.P_OP_MODE_STATE <> iLastOPMode
   //OR  uiLastSeq <> uiSeq
    )
   AND NOT bExitSetReadyState 
THEN
  IF TRUE
  AND fbMainProcess.M_SetReady()
  THEN
    bExitSetReadyState := TRUE;
  ELSE
    RETURN;
  END_IF
END_IF
// Reset set ready state
IF bExitSetReadyState THEN
  bExitSetReadyState := FALSE;
END_IF
iLastOPMode := PrgOrg.fbOpMode.P_OP_MODE_STATE;
uiLastSeq := uiSeq;

IF TRUE
   AND (PrgOrg.fbOpMode.P_EMERGANCY_STOP 
   OR PrgOrg.fbOpMode.P_OP_MODE_STATE = OP_MODE.MACHINE_ERROR 
   OR PrgOrg.fbOpMode.P_OP_MODE_STATE = OP_MODE.SAFETY_STOP) 
THEN
  uiSeq := 10;
ELSIF TRUE
      AND PrgOrg.fbOpMode.P_OP_MODE_STATE = OP_MODE.INIT 
      AND uiSeq = 999
THEN
  bBusyInit := TRUE;
  uiSeq := 20;
ELSIF TRUE 
      AND PrgOrg.fbOpMode.P_OP_MODE_STATE = OP_MODE.STOP 
      AND uiSeq < 999
      AND NOT bBusyStop
THEN
  bBusyStop := TRUE;
  uiSeq := 30;
ELSIF TRUE 
      AND PrgOrg.fbOpMode.P_OP_MODE_STATE = OP_MODE.AUTO 
      //AND PrgOrg.fbOpMode.P_INIT_OK
      AND PrgOrg.bInitOK
      AND PrgVisu.fbVisuOPMode.P_EnduranceRunSelected 
      AND uiSeq = 999
THEN
  uiSeq := 40;
ELSIF TRUE
      AND PrgOrg.fbOpMode.P_OP_MODE_STATE = OP_MODE.AUTO 
      //AND PrgOrg.fbOpMode.P_INIT_OK
      AND PrgOrg.bInitOK
      AND PrgVisu.fbVisuOPMode.P_BreakPressureDetSelected 
      AND uiSeq = 999
THEN
  uiSeq := 50;
ELSIF TRUE 
      AND PrgOrg.fbOpMode.P_OP_MODE_STATE = OP_MODE.AUTO 
      //AND PrgOrg.fbOpMode.P_INIT_OK
      AND PrgOrg.bInitOK
      AND PrgVisu.fbVisuOPMode.P_LeakTest1Selected 
      AND uiSeq = 999
THEN
  uiSeq := 60;
ELSIF TRUE 
      AND PrgOrg.fbOpMode.P_OP_MODE_STATE = OP_MODE.AUTO 
      //AND PrgOrg.fbOpMode.P_INIT_OK
      AND PrgOrg.bInitOK
      AND PrgVisu.fbVisuOPMode.P_LeakTest2Selected 
      AND uiSeq = 999
THEN
  uiSeq := 70;
END_IF

CASE uiSeq OF
  0:  // Base step
    uiSeq := 0;
    
  10: // Emergancy stop or Error
    IF fbMainProcess.M_EStop() THEN
      PrgOrg.bInitOK := FALSE;
      PrgOrg.fbLockDoor.M_Reset();
      uiSeq := 100;
		END_IF
  
  20: // Init
    IF PrgStation.fbMainProcess.M_Reset() THEN
      PrgOrg.bInitOK := TRUE;
      uiSeq := 100;
	  END_IF
      
  30: // Stop
    IF PrgStation.fbMainProcess.M_Stop() THEN
      PrgOrg.bInitOK := FALSE;
      uiSeq := 100;
		END_IF
  
  40: // Auto -> Endurance run
    IF PrgStation.fbMainProcess.M_EnduranceRun(stEnduranceRunParams:= PrgStation.stRecipeParams.stRecipeEnduranceRun) THEN
      uiSeq := 100;
	  END_IF
  
  50: // Auto -> Break pressure detection
    IF PrgStation.fbMainProcess.M_BreakPressureDet(stBreakPressureParams:= PrgStation.stRecipeParams.stRecipeBreakPressure) THEN
      uiSeq := 100;
	  END_IF
  
  60: // Auto -> Leaktest 1
    IF PrgStation.fbMainProcess.M_LeakTest1(stLeakTest1Params:= PrgStation.stRecipeParams.stRecipeLeakTest1) THEN
      uiSeq := 100;
	  END_IF
  
  70: // Auto -> Leaktest 2
    IF PrgStation.fbMainProcess.M_LeakTest2(stLeakTest2Params:= PrgStation.stRecipeParams.stRecipeLeakTest2) THEN
      uiSeq := 100;
	  END_IF
  
  80:
    uiSeq := 0;
  
  90:
    uiSeq := 0;
  
  100:
    PrgOrg.fbOpMode.M_OP_MODE_OFF();
    IF PrgVisu.fbVisuOPMode.M_ResetModeSelection() THEN
      bBusyStop := FALSE;
      bBusyInit := FALSE;
      uiSeq := 999;
    END_IF
END_CASE
END_ACTION

END_PROGRAM

// ---- ORGANISATION/DATE_TIME/POU/FB_CLOCK.TcPOU
FUNCTION_BLOCK FB_CLOCK IMPLEMENTS I_CLOCK
VAR_INPUT
END_VAR
VAR_OUTPUT
END_VAR
VAR
  fbFormat:                   FB_FormatString;
  bError:                     BOOL;
  nErrID:                     UDINT;
  bStart:                     BOOL;
  bPause:                     BOOL;
  fbTimer:                    TON;
  tTimerValue:                TIME;
  fbTrigger:                  R_TRIG;
  tTimeReturn1:               TIME;
  tTimeReturn2:               TIME;
  tPausedTime:                TIME;
  tDifference:                TIME;
  strDifference:              STRING(12);
  uiHours:                    UINT;
  udiMinutes:                 UDINT;
  uliSeconds:                 ULINT;
  uliTotalMilliseconds:       ULINT;
END_VAR

// Timer
fbTimer(IN := bStart, PT := tTimerValue);
fbTrigger(CLK := fbTimer.IN);

IF fbTrigger.Q THEN
    tTimeReturn1  := TIME();
END_IF

IF bStart THEN
  tTimeReturn2  := TIME();
  tDifference   := tTimeReturn2 - tTimeReturn1;
END_IF

IF fbTimer.Q THEN
    //bStart        := FALSE;
END_IF

METHOD M_GetTimerET : STRING
VAR_INPUT
  /// Default: hhh:mm:ss
  bCustomFormat:      BOOL;
  /// Timeformat: mm/ss or hh-mm-ss or dd/hh/mm/ss
  sFormat:            STRING;
END_VAR


// Rechne die Zeit in Millisekunden um
THIS^.uliTotalMilliseconds := TIME_TO_ULINT(THIS^.tDifference);

// Extrahiere Stunden, Minuten und Sekunden
THIS^.uiHours := TO_UINT(THIS^.uliTotalMilliseconds / 3600000);
THIS^.udiMinutes := TO_UDINT((THIS^.uliTotalMilliseconds MOD 3600000) / 60000);
THIS^.uliSeconds := (THIS^.uliTotalMilliseconds MOD 60000) / 1000;

THIS^.fbFormat(sFormat:= '%.3d:%.2d:%.2d', 
               arg1 := F_UINT(THIS^.uiHours), 
               arg2 := F_UDINT(THIS^.udiMinutes), 
               arg3 := F_ULINT(THIS^.uliSeconds), 
               sOut => M_GetTimerET, 
               bError => THIS^.bError, 
               nErrID => THIS^.nErrID);
END_METHOD

{warning 'Methodenimplementierung hinzufügen'}
METHOD M_PauseTimer : BOOL
END_METHOD

{warning 'Methodenimplementierung hinzufügen'}
(*=== Method: M_Run  ============================================

 @brief: Here is the global code (Timer, Event, Flange,...)*)
METHOD M_Run
END_METHOD

METHOD M_StartTimer : BOOL
M_StartTimer := THIS^.tTimerValue = T#49D17H2M47S295MS AND THIS^.bStart = TRUE;

THIS^.tTimerValue := T#49D17H2M47S295MS;
THIS^.bStart := TRUE;
END_METHOD

METHOD M_StopTimer : BOOL
M_StopTimer := THIS^.tTimerValue = T#49D17H2M47S295MS AND THIS^.bStart = FALSE;

THIS^.tTimerValue := T#49D17H2M47S295MS;
THIS^.bStart := FALSE;
END_METHOD

{warning 'Methodenimplementierung hinzufügen'}
METHOD M_WaitForTimer : BOOL
END_METHOD

{warning 'Eigenschaftenimplementierung hinzufügen'}
(*=== Property: P_Event  ============================================

 @param [set]: 	Set the Structure "ST_EVENT" from another Object
 @param [get]: 	Return the Structure "ST_EVENT", it contains the actual 
					event of the Object *)
PROPERTY P_Event : GenLib.ST_EVENT
GET
END_GET
SET
END_SET
END_PROPERTY

{warning 'Eigenschaftenimplementierung hinzufügen'}
(*=== Property: P_FullObjectPath  ============================================

 @param [set]: 	Set the Object Path (Clear String of Object)
 @param [get]: 	Return the Objectpath *)
PROPERTY P_FullObjectPath : STRING
GET
END_GET
SET
END_SET
END_PROPERTY

{warning 'Eigenschaftenimplementierung hinzufügen'}
(*=== Property: P_Global_Ack  ============================================

 @param [set]: 	Set the Bit for Ack from another Object
 @param [get]: 	Return the state of Ack Bit*)
PROPERTY P_Global_Ack : BOOL
GET
END_GET
SET
END_SET
END_PROPERTY

{warning 'Eigenschaftenimplementierung hinzufügen'}
(*=== Property: P_GlobalID  ============================================

 @param [set]: 	-
 @param [get]: 	Return the string of instance path*)
PROPERTY P_GlobalID : STRING
GET
END_GET
END_PROPERTY

{warning 'Eigenschaftenimplementierung hinzufügen'}
PROPERTY P_SystemTime : STRING
GET
END_GET
END_PROPERTY

END_FUNCTION_BLOCK

// ---- MODULE/ACTOR_VALVE/HYDRAULIC_ACTOR/POU/FB_PUMP_WITH_BYPASS.TcPOU
FUNCTION_BLOCK FB_PUMP_WITH_BYPASS IMPLEMENTS I_PUMP_WITH_BYPASS
VAR //General
	{attribute 'instance-path'} 
  {attribute 'noinit'} 
	strInstancePath:									                      STRING;
	bInit: 												                          BOOL:=TRUE;
	strFullObjectPath: 								                      STRING;
	stEvent:											                          ST_EVENT;
	bAck:												                            BOOL;	
END_VAR
VAR   // From FB_init	
  itfOpMode:											                        I_OP_MODE; 
  itfEventLogger:                                         I_EVENT_LOGGER;
  itfOn:                                                  I_BINARY_OUTPUT;
  itfBypassValve:                                         I_VALVE_X_2;
END_VAR                                      				
VAR	// Step chain control                				
  eSeq, eLastSeq, eNextSeq:					                      E_SEQ_ENGINE; 
                  				
  //eActiveSeqState, eLastActiveSeqState:                 E_SEQ_GENERAL;
	(*
  iInternalSeqStateCase, iLastInternalSeqStateCase:       INT:=0;       
	tonDelay, tonTimeOut, tonStepTime:						          TON;
	tDelay:													                        TIME := T#100MS;
	tTimeOut:												                        TIME := T#100MS;
	tTimeOutExt:											                      TIME := T#100MS;
	bDelayActive, bTimeOutActiveQuit, bTimeOutActiveNoQuit:	BOOL;//Timer Option
	bActiveStep, bDebugAcitve, bDebugNext:					        BOOL;//Debug Option
	i:														                          INT;
 	iError:													                        INT; //ERROR-CODE                    	                   		
	listLastSteps:											                    ARRAY[0..49] OF ST_LAST_STEPS;	
	strExtraInfo:											                      STRING; 
	eStep_Type:												                      E_STEP_STATE_TYPE; 
	bDebugModeActive:										                    BOOL;   
	bWaitForBreakpoint:										                  BOOL;
	bBreakpointActive:										                  BOOL;
	bDebugResume:											                      BOOL;   
	listBreakpoint:											                    ARRAY[0..10] OF  INT;    
*)
i:														                            INT;
stSeqCtrlGeneral:											                    ST_SEQ_CTRL_GEN;     	
END_VAR                                             		
VAR                                                 		
	bMethodeFromExtStarted:									                BOOL;
	bMethodeFromExtActive:									                BOOL;
	bMethodeFromExtDone:									                  BOOL;
	strTemp:												                        STRING;
END_VAR   
VAR
  rLimit:                                                 REAL;
  bEnableBypass:                                          BOOL := TRUE;
END_VAR                  	
VAR_TEMP                    	
	iTemp:										                              INT;
END_VAR

// Set FBs and Interfaces ready after switch internal step
IF stSeqCtrlGeneral.iInternalSeqStateCase <> stSeqCtrlGeneral.iLastInternalSeqStateCase AND NOT stSeqCtrlGeneral.bExitSetReadyState THEN
  IF TRUE
  AND itfBypassValve.M_SetReady()
  THEN
    stSeqCtrlGeneral.bExitSetReadyState := TRUE;
  ELSE
    RETURN;
  END_IF
END_IF

stSeqCtrlGeneral.strObject := F_CreateObjectName(strInstancePath);

// First method call
_m_SequenceManager();
//_m_SaveLastStep();

CASE eSeq OF 
  E_SEQ_VALVE.BASE:;
  
	E_SEQ_ENGINE.INIT: _m_Seq_INIT();
		IF TRUE
		AND (stSeqCtrlGeneral.eActiveSeqState = E_SEQ_GENERAL.DONE) 
		THEN
			eSeq := E_SEQ_ENGINE.BASE;
		END_IF
		
	E_SEQ_ENGINE.SETUP:;
  
	// Process
  E_SEQ_ENGINE.ON: _m_Seq_ON();
    IF TRUE
		AND (stSeqCtrlGeneral.eActiveSeqState = E_SEQ_GENERAL.DONE) 
		THEN
			eSeq := E_SEQ_VALVE.BASE;
		END_IF
    
  E_SEQ_ENGINE.OFF: _m_Seq_OFF();
    IF TRUE
		AND (stSeqCtrlGeneral.eActiveSeqState = E_SEQ_GENERAL.DONE) 
		THEN
			eSeq := E_SEQ_VALVE.BASE;
		END_IF
    
  E_SEQ_ENGINE.BYPASS: _m_Seq_BYPASS();
    IF TRUE
		AND (stSeqCtrlGeneral.eActiveSeqState = E_SEQ_GENERAL.DONE) 
		THEN
			eSeq := E_SEQ_VALVE.BASE;
		END_IF

  // End
	E_SEQ_ENGINE.END:;
	E_SEQ_ENGINE.ERROR_SEQ:;	
END_CASE

strTemp:=TO_STRING(eSeq);

METHOD PRIVATE _m_DebugManager
VAR_INPUT
	iStepID: int;
END_VAR
IF TRUE
AND THIS^.stSeqCtrlGeneral.bDebugModeActive 
AND NOT THIS^.stSeqCtrlGeneral.bActiveStep
THEN


THIS^.stSeqCtrlGeneral.bBreakpointActive:=FALSE;

FOR i:=0 TO 10 DO
	
	IF TRUE
	AND iStepID=THIS^.stSeqCtrlGeneral.listBreakpoint[i] 
	AND iStepID<>0
	THEN
		EXIT;
	END_IF
END_FOR
IF (i<=10) THEN
	THIS^.stSeqCtrlGeneral.bBreakpointActive:=TRUE;
END_IF

END_IF
END_METHOD

METHOD PRIVATE _m_Delay : BOOL
VAR_INPUT
	DelayTime:	TIME;
END_VAR
THIS^.stSeqCtrlGeneral.bDelayActive:=TRUE;
THIS^.stSeqCtrlGeneral.tDelay:=DelayTime;
_m_Delay:=FALSE;
IF THIS^.stSeqCtrlGeneral.tonDelay.Q THEN
	_m_Delay:=TRUE;
END_IF
END_METHOD

METHOD PRIVATE _m_GeneralStepSetting : BOOL
VAR_INPUT
	StepType:			    	E_STEP_STATE_TYPE;
	InfoTextID:					STRING(20);
	EnableDebug:	   			BOOL;	
	
END_VAR
IF THIS^.stSeqCtrlGeneral.bActiveStep THEN
	THIS^.stSeqCtrlGeneral.eStep_Type:=StepType;
	THIS^.stSeqCtrlGeneral.strExtraInfo:= GenLib.F_RET_TXTLIST_ENTRY(strPortNr:='851',strID:='',strTxtLstName:=InfoTextID);
END_IF
END_METHOD

METHOD PRIVATE _m_SaveLastStep : BOOL
VAR_INPUT
END_VAR
VAR
	i: dint;
END_VAR
IF NOT THIS^.stSeqCtrlGeneral.bActiveStep THEN
	
	FOR i:=49 TO 1 BY -1 DO
			stSeqCtrlGeneral.listLastSteps[i].strStepName:=stSeqCtrlGeneral.listLastSteps[i-1].strStepName;
			stSeqCtrlGeneral.listLastSteps[i].tStepTime:=stSeqCtrlGeneral.listLastSteps[i-1].tStepTime;
			stSeqCtrlGeneral.listLastSteps[i].tDelayTime:=stSeqCtrlGeneral.listLastSteps[i-1].tDelayTime;
	END_FOR
	stSeqCtrlGeneral.listLastSteps[0].strStepName:=TO_STRING(THIS^.eSeq);
	stSeqCtrlGeneral.listLastSteps[1].tStepTime:=THIS^.stSeqCtrlGeneral.tonStepTime.ET;
	stSeqCtrlGeneral.listLastSteps[1].tStepTime:=THIS^.stSeqCtrlGeneral.tonDelay.ET;
ELSE
	stSeqCtrlGeneral.listLastSteps[0].tStepTime:=THIS^.stSeqCtrlGeneral.tonStepTime.ET;
	stSeqCtrlGeneral.listLastSteps[0].tDelayTime:=THIS^.stSeqCtrlGeneral.tonDelay.ET;	
END_IF
END_METHOD

METHOD PRIVATE _m_Seq_BYPASS : BOOL
VAR
  ActiveSeq: STRING;
END_VAR
//THIS^._m_GeneralStepSetting(StepType:=E_STEP_STATE_TYPE.INIT,
ActiveSeq := TO_STRING(THIS^.eSeq);

CASE THIS^.stSeqCtrlGeneral.eActiveSeqState OF
E_SEQ_GENERAL.READY:;
	
E_SEQ_GENERAL.EXECUTE:;
	IF TRUE
	THEN
		THIS^.stSeqCtrlGeneral.eActiveSeqState := E_SEQ_GENERAL.RESET;
	END_IF
  
E_SEQ_GENERAL.RESET:;
	stSeqCtrlGeneral.iInternalSeqStateCase := 0;
	IF TRUE
	THEN
		THIS^.stSeqCtrlGeneral.eActiveSeqState := E_SEQ_GENERAL.BUSY;
	END_IF
  
E_SEQ_GENERAL.BUSY:;
	CASE THIS^.stSeqCtrlGeneral.iInternalSeqStateCase OF
    0:  // Bypass
      IF TRUE 
      AND THIS^.bEnableBypass
			THEN 
        IF THIS^.itfBypassValve.M_ToHP(tDelay:= T#10MS) THEN
          THIS^.stSeqCtrlGeneral.iInternalSeqStateCase := 1000;
				END_IF
      ELSE
        IF THIS^.itfBypassValve.M_ToWP1(tDelay:= T#10MS) THEN
          THIS^.stSeqCtrlGeneral.iInternalSeqStateCase := 1000;
        END_IF
			END_IF
      
	ELSE
		THIS^.stSeqCtrlGeneral.eActiveSeqState := E_SEQ_GENERAL.DONE;  
	END_CASE
	THIS^.stSeqCtrlGeneral.strExtraInfo := CONCAT('Internal state: ', TO_STRING(THIS^.stSeqCtrlGeneral.iInternalSeqStateCase));

E_SEQ_GENERAL.DONE:;

E_SEQ_GENERAL.ERROR:;

E_SEQ_GENERAL.TIME_OUT:; 
IF TRUE
AND THIS^.stSeqCtrlGeneral.bTimeOutActiveQuit 
THEN
  THIS^.stSeqCtrlGeneral.strExtraInfo := 'Bitte quittieren und erneut testen';
  IF TRUE
  //AND itfOpMode.P_QUIT
  THEN
    THIS^.stSeqCtrlGeneral.eActiveSeqState := E_SEQ_GENERAL.EXECUTE;
	END_IF
  
END_IF

ELSE
  THIS^.stSeqCtrlGeneral.eActiveSeqState := E_SEQ_GENERAL.ERROR;
END_CASE
END_METHOD

METHOD PRIVATE _m_Seq_INIT : BOOL
VAR
  ActiveSeq: STRING;
END_VAR
//THIS^._m_GeneralStepSetting(StepType:=E_STEP_STATE_TYPE.INIT,
ActiveSeq := TO_STRING(THIS^.eSeq);

CASE THIS^.stSeqCtrlGeneral.eActiveSeqState OF
E_SEQ_GENERAL.READY:;

	
E_SEQ_GENERAL.EXECUTE:;
	IF TRUE
	THEN
		THIS^.stSeqCtrlGeneral.eActiveSeqState := E_SEQ_GENERAL.RESET;
	END_IF
  
E_SEQ_GENERAL.RESET:;
	stSeqCtrlGeneral.iInternalSeqStateCase := 0;
	IF TRUE
	THEN
		THIS^.stSeqCtrlGeneral.eActiveSeqState := E_SEQ_GENERAL.BUSY;
	END_IF
  
E_SEQ_GENERAL.BUSY:;
	CASE THIS^.stSeqCtrlGeneral.iInternalSeqStateCase OF
    0:  // Reset engine
      IF TRUE 
			THEN 
        THIS^.itfOn.M_Reset();
        THIS^.stSeqCtrlGeneral.iInternalSeqStateCase := 10;
			END_IF
    
    10: // Enable bypass
      IF TRUE 
      AND THIS^.itfBypassValve.M_ToHP(tDelay:= T#10MS)
			THEN 
        THIS^.stSeqCtrlGeneral.iInternalSeqStateCase := 1000;
			END_IF
      
	ELSE
		THIS^.stSeqCtrlGeneral.eActiveSeqState := E_SEQ_GENERAL.DONE;  
	END_CASE
	THIS^.stSeqCtrlGeneral.strExtraInfo := CONCAT('Internal state: ', TO_STRING(THIS^.stSeqCtrlGeneral.iInternalSeqStateCase));

E_SEQ_GENERAL.DONE:;

E_SEQ_GENERAL.ERROR:;

E_SEQ_GENERAL.TIME_OUT:; 
IF TRUE
AND THIS^.stSeqCtrlGeneral.bTimeOutActiveQuit 
THEN
  THIS^.stSeqCtrlGeneral.strExtraInfo := 'Bitte quittieren und erneut testen';
  IF TRUE
  //AND itfOpMode.P_QUIT
  THEN
    THIS^.stSeqCtrlGeneral.eActiveSeqState := E_SEQ_GENERAL.EXECUTE;
	END_IF
  
END_IF

ELSE
  THIS^.stSeqCtrlGeneral.eActiveSeqState := E_SEQ_GENERAL.ERROR;
END_CASE
END_METHOD

METHOD _m_Seq_OFF : BOOL
VAR
  ActiveSeq: STRING;
END_VAR
//THIS^._m_GeneralStepSetting(StepType:=E_STEP_STATE_TYPE.INIT,
ActiveSeq := TO_STRING(THIS^.eSeq);

CASE THIS^.stSeqCtrlGeneral.eActiveSeqState OF
E_SEQ_GENERAL.READY:;

	
E_SEQ_GENERAL.EXECUTE:;
	IF TRUE
	THEN
		THIS^.stSeqCtrlGeneral.eActiveSeqState := E_SEQ_GENERAL.RESET;
	END_IF
  
E_SEQ_GENERAL.RESET:;
	stSeqCtrlGeneral.iInternalSeqStateCase := 0;
	IF TRUE
	THEN
		THIS^.stSeqCtrlGeneral.eActiveSeqState := E_SEQ_GENERAL.BUSY;
	END_IF
  
E_SEQ_GENERAL.BUSY:;
	CASE THIS^.stSeqCtrlGeneral.iInternalSeqStateCase OF
    0:  // Engine off
      IF TRUE 
			THEN 
        THIS^.itfOn.M_Reset();
        THIS^.stSeqCtrlGeneral.iInternalSeqStateCase := 1000;
			END_IF
      
	ELSE
		THIS^.stSeqCtrlGeneral.eActiveSeqState := E_SEQ_GENERAL.DONE;  
	END_CASE
	THIS^.stSeqCtrlGeneral.strExtraInfo := CONCAT('Internal state: ', TO_STRING(THIS^.stSeqCtrlGeneral.iInternalSeqStateCase));

E_SEQ_GENERAL.DONE:;

E_SEQ_GENERAL.ERROR:;

E_SEQ_GENERAL.TIME_OUT:; 
IF TRUE
AND THIS^.stSeqCtrlGeneral.bTimeOutActiveQuit 
THEN
  THIS^.stSeqCtrlGeneral.strExtraInfo := 'Bitte quittieren und erneut testen';
  IF TRUE
  //AND itfOpMode.P_QUIT
  THEN
    THIS^.stSeqCtrlGeneral.eActiveSeqState := E_SEQ_GENERAL.EXECUTE;
	END_IF
  
END_IF

ELSE
  THIS^.stSeqCtrlGeneral.eActiveSeqState := E_SEQ_GENERAL.ERROR;
END_CASE
END_METHOD

METHOD PRIVATE _m_Seq_ON : BOOL
VAR
  ActiveSeq: STRING;
END_VAR
//THIS^._m_GeneralStepSetting(StepType:=E_STEP_STATE_TYPE.INIT,
ActiveSeq := TO_STRING(THIS^.eSeq);

CASE THIS^.stSeqCtrlGeneral.eActiveSeqState OF
E_SEQ_GENERAL.READY:;

	
E_SEQ_GENERAL.EXECUTE:;
	IF TRUE
	THEN
		THIS^.stSeqCtrlGeneral.eActiveSeqState := E_SEQ_GENERAL.RESET;
	END_IF
  
E_SEQ_GENERAL.RESET:;
	stSeqCtrlGeneral.iInternalSeqStateCase := 0;
	IF TRUE
	THEN
		THIS^.stSeqCtrlGeneral.eActiveSeqState := E_SEQ_GENERAL.BUSY;
	END_IF
  
E_SEQ_GENERAL.BUSY:;
	CASE THIS^.stSeqCtrlGeneral.iInternalSeqStateCase OF
    0:  // Engine on
      IF TRUE 
			THEN 
        THIS^.itfOn.M_Set();
        THIS^.stSeqCtrlGeneral.iInternalSeqStateCase := 1000;
			END_IF
      
	ELSE
		THIS^.stSeqCtrlGeneral.eActiveSeqState := E_SEQ_GENERAL.DONE;  
	END_CASE
	THIS^.stSeqCtrlGeneral.strExtraInfo := CONCAT('Internal state: ', TO_STRING(THIS^.stSeqCtrlGeneral.iInternalSeqStateCase));

E_SEQ_GENERAL.DONE:;

E_SEQ_GENERAL.ERROR:;

E_SEQ_GENERAL.TIME_OUT:; 
IF TRUE
AND THIS^.stSeqCtrlGeneral.bTimeOutActiveQuit 
THEN
  THIS^.stSeqCtrlGeneral.strExtraInfo := 'Bitte quittieren und erneut testen';
  IF TRUE
  //AND itfOpMode.P_QUIT
  THEN
    THIS^.stSeqCtrlGeneral.eActiveSeqState := E_SEQ_GENERAL.EXECUTE;
	END_IF
  
END_IF

ELSE
  THIS^.stSeqCtrlGeneral.eActiveSeqState := E_SEQ_GENERAL.ERROR;
END_CASE
END_METHOD

METHOD PRIVATE _m_SequenceManager
VAR_INPUT
END_VAR
IF FALSE
//AND THIS^.eActiveSeqState=DONE 
AND eLastSeq<>eSeq
THEN
	IF THIS^.stSeqCtrlGeneral.eActiveSeqState<>E_SEQ_GENERAL.EXECUTE THEN
		THIS^.stSeqCtrlGeneral.eActiveSeqState:=E_SEQ_GENERAL.READY;
	END_IF
END_IF

eSeq := eNextSeq;

//DelayTimer und TimeOut Timer verwalten
stSeqCtrlGeneral.bActiveStep:=	TRUE
				AND eLastSeq					=	eSeq
				AND stSeqCtrlGeneral.eLastActiveSeqState			=	stSeqCtrlGeneral.eActiveSeqState
				AND	stSeqCtrlGeneral.iLastInternalSeqStateCase	=	stSeqCtrlGeneral.iInternalSeqStateCase
				;
			
IF NOT stSeqCtrlGeneral.bActiveStep THEN
	stSeqCtrlGeneral.bDelayActive:=FALSE;
	stSeqCtrlGeneral.bTimeOutActiveQuit:=FALSE;
	stSeqCtrlGeneral.bTimeOutActiveNoQuit:=FALSE;
  THIS^.stSeqCtrlGeneral.strExtraInfo:='';
END_IF

_m_SaveLastStep();
stSeqCtrlGeneral.tonDelay	(IN:=stSeqCtrlGeneral.bActiveStep AND stSeqCtrlGeneral.bDelayActive, 		PT:=stSeqCtrlGeneral.tDelay);
stSeqCtrlGeneral.tonTimeOut	(IN:=stSeqCtrlGeneral.bActiveStep AND (stSeqCtrlGeneral.bTimeOutActiveNoQuit OR stSeqCtrlGeneral.bTimeOutActiveQuit), 	PT:=stSeqCtrlGeneral.tTimeOut);
stSeqCtrlGeneral.tonStepTime	(IN:= stSeqCtrlGeneral.bActiveStep, PT:= T#24H);

IF stSeqCtrlGeneral.tonTimeOut.Q  THEN
	stSeqCtrlGeneral.eActiveSeqState:=E_SEQ_GENERAL.TIME_OUT;
END_IF

IF stSeqCtrlGeneral.iError<>0 THEN
	eSeq:=E_SEQ_ENGINE.ERROR_SEQ;
END_IF



eLastSeq					:=	eSeq;
stSeqCtrlGeneral.eLastActiveSeqState			:=	stSeqCtrlGeneral.eActiveSeqState;
stSeqCtrlGeneral.iLastInternalSeqStateCase	:=	stSeqCtrlGeneral.iInternalSeqStateCase;

// Reset set ready state
IF THIS^.stSeqCtrlGeneral.bExitSetReadyState THEN
  THIS^.stSeqCtrlGeneral.bExitSetReadyState := FALSE;
END_IF
END_METHOD

METHOD PRIVATE _m_TimeOut : BOOL
VAR_INPUT
	bTimeoutActiveToQuit:	BOOL;
	bTimeOutActiveNoQuit:	BOOL;
	tTimeOut:				TIME;	
END_VAR
THIS^.stSeqCtrlGeneral.bTimeOutActiveQuit:=	bTimeoutActiveToQuit;
THIS^.stSeqCtrlGeneral.bTimeOutActiveNoQuit:=	bTimeOutActiveNoQuit;
THIS^.stSeqCtrlGeneral.tTimeOut:=			tTimeOut;
_m_TimeOut:=FALSE;
IF THIS^.stSeqCtrlGeneral.tonTimeOut.Q THEN
	_m_TimeOut:=TRUE;
END_IF
END_METHOD

METHOD FB_init : BOOL
VAR_INPUT
	bInitRetains : BOOL; // if TRUE, the retain variables are initialized (warm start / cold start)
	bInCopyCode : BOOL;  // if TRUE, the instance afterwards gets moved into the copy code (online change)
  
  itfOpMode:											                        I_OP_MODE; 
  itfEventLogger:                                         I_EVENT_LOGGER;
  itfOn:                                                  I_BINARY_OUTPUT;
  itfBypassValve:                                         I_VALVE_X_2;
END_VAR
THIS^.itfOpMode := itfOpMode;
THIS^.itfEventLogger := itfEventLogger;
THIS^.itfOn := itfOn;
THIS^.itfBypassValve := itfBypassValve;
END_METHOD

METHOD M_Bypass : BOOL
VAR_INPUT
  bEnable:        BOOL;
END_VAR
M_Bypass := THIS^.stSeqCtrlGeneral.eActiveSeqState = E_SEQ_GENERAL.DONE;

// Assign input
  THIS^.bEnableBypass := bEnable;

// General
IF THIS^.stSeqCtrlGeneral.eActiveSeqState = E_SEQ_GENERAL.READY THEN
  THIS^.eNextSeq := E_SEQ_ENGINE.BYPASS;
  THIS^.stSeqCtrlGeneral.eActiveSeqState := E_SEQ_GENERAL.EXECUTE;
END_IF
END_METHOD

METHOD M_Off : BOOL
M_Off := THIS^.stSeqCtrlGeneral.eActiveSeqState = E_SEQ_GENERAL.DONE;

// Assign input

// General
IF THIS^.stSeqCtrlGeneral.eActiveSeqState = E_SEQ_GENERAL.READY THEN
  THIS^.eNextSeq := E_SEQ_ENGINE.OFF;
  THIS^.stSeqCtrlGeneral.eActiveSeqState := E_SEQ_GENERAL.EXECUTE;
END_IF
END_METHOD

METHOD M_On : BOOL
M_On := THIS^.stSeqCtrlGeneral.eActiveSeqState = E_SEQ_GENERAL.DONE;

// Assign input

// General
IF THIS^.stSeqCtrlGeneral.eActiveSeqState = E_SEQ_GENERAL.READY THEN
  THIS^.eNextSeq := E_SEQ_ENGINE.ON;
  THIS^.stSeqCtrlGeneral.eActiveSeqState := E_SEQ_GENERAL.EXECUTE;
END_IF
END_METHOD

METHOD M_Reset : BOOL
VAR_INPUT
END_VAR
M_Reset := THIS^.stSeqCtrlGeneral.eActiveSeqState = E_SEQ_GENERAL.DONE;

// Assign input

// General
IF THIS^.stSeqCtrlGeneral.eActiveSeqState = E_SEQ_GENERAL.READY THEN
  THIS^.eNextSeq := E_SEQ_ENGINE.INIT;
  THIS^.stSeqCtrlGeneral.eActiveSeqState := E_SEQ_GENERAL.EXECUTE;
END_IF
END_METHOD

{warning 'Methodenimplementierung hinzufügen'}
(*=== Method: M_Run  ============================================

 @brief: Here is the global code (Timer, Event, Flange,...)*)
METHOD M_Run
END_METHOD

METHOD M_SetReady : BOOL
VAR_INPUT
END_VAR
M_SetReady := TRUE
              AND THIS^.stSeqCtrlGeneral.eActiveSeqState = E_SEQ_GENERAL.READY
              AND THIS^.eSeq = E_SEQ_ENGINE.BASE;

THIS^.stSeqCtrlGeneral.eActiveSeqState := E_SEQ_GENERAL.READY;
THIS^.eNextSeq := E_SEQ_ENGINE.BASE;
END_METHOD

{warning 'Eigenschaftenimplementierung hinzufügen'}
PROPERTY P_Busy : BOOL
GET
IF stSeqCtrlGeneral.eActiveSeqState = E_SEQ_GENERAL.READY THEN
  P_Busy := FALSE;
ELSE
  P_Busy := TRUE;
END_IF
END_GET
END_PROPERTY

{warning 'Eigenschaftenimplementierung hinzufügen'}
PROPERTY P_BypassState : BOOL
GET
P_BypassState := itfBypassValve.P_InWP1;
END_GET
END_PROPERTY

{warning 'Eigenschaftenimplementierung hinzufügen'}
(*=== Property: P_Event  ============================================

 @param [set]: 	Set the Structure "ST_EVENT" from another Object
 @param [get]: 	Return the Structure "ST_EVENT", it contains the actual 
					event of the Object *)
PROPERTY P_Event : GenLib.ST_EVENT
GET
END_GET
SET
END_SET
END_PROPERTY

{warning 'Eigenschaftenimplementierung hinzufügen'}
(*=== Property: P_FullObjectPath  ============================================

 @param [set]: 	Set the Object Path (Clear String of Object)
 @param [get]: 	Return the Objectpath *)
PROPERTY P_FullObjectPath : STRING
GET
END_GET
SET
END_SET
END_PROPERTY

{warning 'Eigenschaftenimplementierung hinzufügen'}
(*=== Property: P_Global_Ack  ============================================

 @param [set]: 	Set the Bit for Ack from another Object
 @param [get]: 	Return the state of Ack Bit*)
PROPERTY P_Global_Ack : BOOL
GET
END_GET
SET
END_SET
END_PROPERTY

{warning 'Eigenschaftenimplementierung hinzufügen'}
(*=== Property: P_GlobalID  ============================================

 @param [set]: 	-
 @param [get]: 	Return the string of instance path*)
PROPERTY P_GlobalID : STRING
GET
END_GET
END_PROPERTY

{warning 'Eigenschaftenimplementierung hinzufügen'}
PROPERTY P_ReadyState : BOOL
GET
P_ReadyState := THIS^.stSeqCtrlGeneral.eActiveSeqState = E_SEQ_GENERAL.READY;
END_GET
END_PROPERTY

{warning 'Eigenschaftenimplementierung hinzufügen'}
PROPERTY P_State : BOOL
GET
P_State := itfOn.P_State;
END_GET
END_PROPERTY

END_FUNCTION_BLOCK

// ---- MODULE/ACTOR_VALVE/HYDRAULIC_ACTOR/POU/FB_PUMP.TcPOU
FUNCTION_BLOCK FB_PUMP IMPLEMENTS I_PUMP
VAR //General
	{attribute 'instance-path'} 
  {attribute 'noinit'} 
	strInstancePath:									                      STRING;
	bInit: 												                          BOOL:=TRUE;
	strFullObjectPath: 								                      STRING;
	stEvent:											                          ST_EVENT;
	bAck:												                            BOOL;	
END_VAR
VAR   // From FB_init	
	itfOpMode:											                        I_OP_MODE; 
  itfEventLogger:                                         I_EVENT_LOGGER;
  itfOn:                                                  I_BINARY_OUTPUT;
END_VAR                                      				
VAR	// Step chain control                				
  eSeq, eLastSeq, eNextSeq:					                      E_SEQ_ENGINE; 
                  				
  //eActiveSeqState, eLastActiveSeqState:                 E_SEQ_GENERAL;
	(*
  iInternalSeqStateCase, iLastInternalSeqStateCase:       INT:=0;       
	tonDelay, tonTimeOut, tonStepTime:						          TON;
	tDelay:													                        TIME := T#100MS;
	tTimeOut:												                        TIME := T#100MS;
	tTimeOutExt:											                      TIME := T#100MS;
	bDelayActive, bTimeOutActiveQuit, bTimeOutActiveNoQuit:	BOOL;//Timer Option
	bActiveStep, bDebugAcitve, bDebugNext:					        BOOL;//Debug Option
	i:														                          INT;
 	iError:													                        INT; //ERROR-CODE                    	                   		
	listLastSteps:											                    ARRAY[0..49] OF ST_LAST_STEPS;	
	strExtraInfo:											                      STRING; 
	eStep_Type:												                      E_STEP_STATE_TYPE; 
	bDebugModeActive:										                    BOOL;   
	bWaitForBreakpoint:										                  BOOL;
	bBreakpointActive:										                  BOOL;
	bDebugResume:											                      BOOL;   
	listBreakpoint:											                    ARRAY[0..10] OF  INT;    
*)
i:														                            INT;
stSeqCtrlGeneral:											                    ST_SEQ_CTRL_GEN;     	
END_VAR                                             		
VAR                                                 		
	bMethodeFromExtStarted:									                BOOL;
	bMethodeFromExtActive:									                BOOL;
	bMethodeFromExtDone:									                  BOOL;
	strTemp:												                        STRING;
END_VAR   
VAR
  rLimit:                                                 REAL;
END_VAR                  	
VAR_TEMP                    	
	iTemp:										                              INT;
END_VAR

// Set FBs and Interfaces ready after switch internal step
IF stSeqCtrlGeneral.iInternalSeqStateCase <> stSeqCtrlGeneral.iLastInternalSeqStateCase AND NOT stSeqCtrlGeneral.bExitSetReadyState THEN
  IF TRUE
  //AND ...
  THEN
    stSeqCtrlGeneral.bExitSetReadyState := TRUE;
  ELSE
    RETURN;
  END_IF
END_IF

stSeqCtrlGeneral.strObject := F_CreateObjectName(strInstancePath);

// First method call
_m_SequenceManager();
//_m_SaveLastStep();

CASE eSeq OF 
  E_SEQ_VALVE.BASE:;
  
	E_SEQ_ENGINE.INIT: _m_Seq_INIT();
		IF TRUE
		AND (stSeqCtrlGeneral.eActiveSeqState = E_SEQ_GENERAL.DONE) 
		THEN
			eSeq := E_SEQ_ENGINE.BASE;
		END_IF
		
	E_SEQ_ENGINE.SETUP:;
  
	// Process
  E_SEQ_ENGINE.ON: _m_Seq_ON();
    IF TRUE
		AND (stSeqCtrlGeneral.eActiveSeqState = E_SEQ_GENERAL.DONE) 
		THEN
			eSeq := E_SEQ_VALVE.BASE;
		END_IF
    
  E_SEQ_ENGINE.OFF: _m_Seq_OFF();
    IF TRUE
		AND (stSeqCtrlGeneral.eActiveSeqState = E_SEQ_GENERAL.DONE) 
		THEN
			eSeq := E_SEQ_VALVE.BASE;
		END_IF

  // End
	E_SEQ_ENGINE.END:;
	E_SEQ_ENGINE.ERROR_SEQ:;	
END_CASE

strTemp:=TO_STRING(eSeq);

METHOD PRIVATE _m_DebugManager
VAR_INPUT
	iStepID: int;
END_VAR
IF TRUE
AND THIS^.stSeqCtrlGeneral.bDebugModeActive 
AND NOT THIS^.stSeqCtrlGeneral.bActiveStep
THEN


THIS^.stSeqCtrlGeneral.bBreakpointActive:=FALSE;

FOR i:=0 TO 10 DO
	
	IF TRUE
	AND iStepID=THIS^.stSeqCtrlGeneral.listBreakpoint[i] 
	AND iStepID<>0
	THEN
		EXIT;
	END_IF
END_FOR
IF (i<=10) THEN
	THIS^.stSeqCtrlGeneral.bBreakpointActive:=TRUE;
END_IF

END_IF
END_METHOD

METHOD PRIVATE _m_Delay : BOOL
VAR_INPUT
	DelayTime:	TIME;
END_VAR
THIS^.stSeqCtrlGeneral.bDelayActive:=TRUE;
THIS^.stSeqCtrlGeneral.tDelay:=DelayTime;
_m_Delay:=FALSE;
IF THIS^.stSeqCtrlGeneral.tonDelay.Q THEN
	_m_Delay:=TRUE;
END_IF
END_METHOD

METHOD PRIVATE _m_GeneralStepSetting : BOOL
VAR_INPUT
	StepType:			    	E_STEP_STATE_TYPE;
	InfoTextID:					STRING(20);
	EnableDebug:	   			BOOL;	
	
END_VAR
IF THIS^.stSeqCtrlGeneral.bActiveStep THEN
	THIS^.stSeqCtrlGeneral.eStep_Type:=StepType;
	THIS^.stSeqCtrlGeneral.strExtraInfo:= GenLib.F_RET_TXTLIST_ENTRY(strPortNr:='851',strID:='',strTxtLstName:=InfoTextID);
END_IF
END_METHOD

METHOD PRIVATE _m_SaveLastStep : BOOL
VAR_INPUT
END_VAR
VAR
	i: dint;
END_VAR
IF NOT THIS^.stSeqCtrlGeneral.bActiveStep THEN
	
	FOR i:=49 TO 1 BY -1 DO
			stSeqCtrlGeneral.listLastSteps[i].strStepName:=stSeqCtrlGeneral.listLastSteps[i-1].strStepName;
			stSeqCtrlGeneral.listLastSteps[i].tStepTime:=stSeqCtrlGeneral.listLastSteps[i-1].tStepTime;
			stSeqCtrlGeneral.listLastSteps[i].tDelayTime:=stSeqCtrlGeneral.listLastSteps[i-1].tDelayTime;
	END_FOR
	stSeqCtrlGeneral.listLastSteps[0].strStepName:=TO_STRING(THIS^.eSeq);
	stSeqCtrlGeneral.listLastSteps[1].tStepTime:=THIS^.stSeqCtrlGeneral.tonStepTime.ET;
	stSeqCtrlGeneral.listLastSteps[1].tStepTime:=THIS^.stSeqCtrlGeneral.tonDelay.ET;
ELSE
	stSeqCtrlGeneral.listLastSteps[0].tStepTime:=THIS^.stSeqCtrlGeneral.tonStepTime.ET;
	stSeqCtrlGeneral.listLastSteps[0].tDelayTime:=THIS^.stSeqCtrlGeneral.tonDelay.ET;	
END_IF
END_METHOD

METHOD PRIVATE _m_Seq_INIT : BOOL
VAR
  ActiveSeq: STRING;
END_VAR
//THIS^._m_GeneralStepSetting(StepType:=E_STEP_STATE_TYPE.INIT,
ActiveSeq := TO_STRING(THIS^.eSeq);

CASE THIS^.stSeqCtrlGeneral.eActiveSeqState OF
E_SEQ_GENERAL.READY:;

	
E_SEQ_GENERAL.EXECUTE:;
	IF TRUE
	THEN
		THIS^.stSeqCtrlGeneral.eActiveSeqState := E_SEQ_GENERAL.RESET;
	END_IF
  
E_SEQ_GENERAL.RESET:;
	stSeqCtrlGeneral.iInternalSeqStateCase := 0;
	IF TRUE
	THEN
		THIS^.stSeqCtrlGeneral.eActiveSeqState := E_SEQ_GENERAL.BUSY;
	END_IF
  
E_SEQ_GENERAL.BUSY:;
	CASE THIS^.stSeqCtrlGeneral.iInternalSeqStateCase OF
    0:  // Reset engine
      IF TRUE 
			THEN 
        THIS^.itfOn.M_Reset();
        THIS^.stSeqCtrlGeneral.iInternalSeqStateCase := 1000;
			END_IF
      
	ELSE
		THIS^.stSeqCtrlGeneral.eActiveSeqState := E_SEQ_GENERAL.DONE;  
	END_CASE
	THIS^.stSeqCtrlGeneral.strExtraInfo := CONCAT('Internal state: ', TO_STRING(THIS^.stSeqCtrlGeneral.iInternalSeqStateCase));

E_SEQ_GENERAL.DONE:;

E_SEQ_GENERAL.ERROR:;

E_SEQ_GENERAL.TIME_OUT:; 
IF TRUE
AND THIS^.stSeqCtrlGeneral.bTimeOutActiveQuit 
THEN
  THIS^.stSeqCtrlGeneral.strExtraInfo := 'Bitte quittieren und erneut testen';
  IF TRUE
  //AND itfOpMode.P_QUIT
  THEN
    THIS^.stSeqCtrlGeneral.eActiveSeqState := E_SEQ_GENERAL.EXECUTE;
	END_IF
  
END_IF

ELSE
  THIS^.stSeqCtrlGeneral.eActiveSeqState := E_SEQ_GENERAL.ERROR;
END_CASE
END_METHOD

METHOD _m_Seq_OFF : BOOL
VAR
  ActiveSeq: STRING;
END_VAR
//THIS^._m_GeneralStepSetting(StepType:=E_STEP_STATE_TYPE.INIT,
ActiveSeq := TO_STRING(THIS^.eSeq);

CASE THIS^.stSeqCtrlGeneral.eActiveSeqState OF
E_SEQ_GENERAL.READY:;

	
E_SEQ_GENERAL.EXECUTE:;
	IF TRUE
	THEN
		THIS^.stSeqCtrlGeneral.eActiveSeqState := E_SEQ_GENERAL.RESET;
	END_IF
  
E_SEQ_GENERAL.RESET:;
	stSeqCtrlGeneral.iInternalSeqStateCase := 0;
	IF TRUE
	THEN
		THIS^.stSeqCtrlGeneral.eActiveSeqState := E_SEQ_GENERAL.BUSY;
	END_IF
  
E_SEQ_GENERAL.BUSY:;
	CASE THIS^.stSeqCtrlGeneral.iInternalSeqStateCase OF
    0:  // Engine off
      IF TRUE 
			THEN 
        THIS^.itfOn.M_Reset();
        THIS^.stSeqCtrlGeneral.iInternalSeqStateCase := 1000;
			END_IF
      
	ELSE
		THIS^.stSeqCtrlGeneral.eActiveSeqState := E_SEQ_GENERAL.DONE;  
	END_CASE
	THIS^.stSeqCtrlGeneral.strExtraInfo := CONCAT('Internal state: ', TO_STRING(THIS^.stSeqCtrlGeneral.iInternalSeqStateCase));

E_SEQ_GENERAL.DONE:;

E_SEQ_GENERAL.ERROR:;

E_SEQ_GENERAL.TIME_OUT:; 
IF TRUE
AND THIS^.stSeqCtrlGeneral.bTimeOutActiveQuit 
THEN
  THIS^.stSeqCtrlGeneral.strExtraInfo := 'Bitte quittieren und erneut testen';
  IF TRUE
  //AND itfOpMode.P_QUIT
  THEN
    THIS^.stSeqCtrlGeneral.eActiveSeqState := E_SEQ_GENERAL.EXECUTE;
	END_IF
  
END_IF

ELSE
  THIS^.stSeqCtrlGeneral.eActiveSeqState := E_SEQ_GENERAL.ERROR;
END_CASE
END_METHOD

METHOD PRIVATE _m_Seq_ON : BOOL
VAR
  ActiveSeq: STRING;
END_VAR
//THIS^._m_GeneralStepSetting(StepType:=E_STEP_STATE_TYPE.INIT,
ActiveSeq := TO_STRING(THIS^.eSeq);

CASE THIS^.stSeqCtrlGeneral.eActiveSeqState OF
E_SEQ_GENERAL.READY:;

	
E_SEQ_GENERAL.EXECUTE:;
	IF TRUE
	THEN
		THIS^.stSeqCtrlGeneral.eActiveSeqState := E_SEQ_GENERAL.RESET;
	END_IF
  
E_SEQ_GENERAL.RESET:;
	stSeqCtrlGeneral.iInternalSeqStateCase := 0;
	IF TRUE
	THEN
		THIS^.stSeqCtrlGeneral.eActiveSeqState := E_SEQ_GENERAL.BUSY;
	END_IF
  
E_SEQ_GENERAL.BUSY:;
	CASE THIS^.stSeqCtrlGeneral.iInternalSeqStateCase OF
    0:  // Engine on
      IF TRUE 
			THEN 
        THIS^.itfOn.M_Set();
        THIS^.stSeqCtrlGeneral.iInternalSeqStateCase := 1000;
			END_IF
      
	ELSE
		THIS^.stSeqCtrlGeneral.eActiveSeqState := E_SEQ_GENERAL.DONE;  
	END_CASE
	THIS^.stSeqCtrlGeneral.strExtraInfo := CONCAT('Internal state: ', TO_STRING(THIS^.stSeqCtrlGeneral.iInternalSeqStateCase));

E_SEQ_GENERAL.DONE:;

E_SEQ_GENERAL.ERROR:;

E_SEQ_GENERAL.TIME_OUT:; 
IF TRUE
AND THIS^.stSeqCtrlGeneral.bTimeOutActiveQuit 
THEN
  THIS^.stSeqCtrlGeneral.strExtraInfo := 'Bitte quittieren und erneut testen';
  IF TRUE
  //AND itfOpMode.P_QUIT
  THEN
    THIS^.stSeqCtrlGeneral.eActiveSeqState := E_SEQ_GENERAL.EXECUTE;
	END_IF
  
END_IF

ELSE
  THIS^.stSeqCtrlGeneral.eActiveSeqState := E_SEQ_GENERAL.ERROR;
END_CASE
END_METHOD

METHOD PRIVATE _m_SequenceManager
VAR_INPUT
END_VAR
IF FALSE
//AND THIS^.eActiveSeqState=DONE 
AND eLastSeq<>eSeq
THEN
	IF THIS^.stSeqCtrlGeneral.eActiveSeqState<>E_SEQ_GENERAL.EXECUTE THEN
		THIS^.stSeqCtrlGeneral.eActiveSeqState:=E_SEQ_GENERAL.READY;
	END_IF
END_IF

eSeq := eNextSeq;

//DelayTimer und TimeOut Timer verwalten
stSeqCtrlGeneral.bActiveStep:=	TRUE
				AND eLastSeq					=	eSeq
				AND stSeqCtrlGeneral.eLastActiveSeqState			=	stSeqCtrlGeneral.eActiveSeqState
				AND	stSeqCtrlGeneral.iLastInternalSeqStateCase	=	stSeqCtrlGeneral.iInternalSeqStateCase
				;
			
IF NOT stSeqCtrlGeneral.bActiveStep THEN
	stSeqCtrlGeneral.bDelayActive:=FALSE;
	stSeqCtrlGeneral.bTimeOutActiveQuit:=FALSE;
	stSeqCtrlGeneral.bTimeOutActiveNoQuit:=FALSE;
  THIS^.stSeqCtrlGeneral.strExtraInfo:='';
END_IF

_m_SaveLastStep();
stSeqCtrlGeneral.tonDelay	(IN:=stSeqCtrlGeneral.bActiveStep AND stSeqCtrlGeneral.bDelayActive, 		PT:=stSeqCtrlGeneral.tDelay);
stSeqCtrlGeneral.tonTimeOut	(IN:=stSeqCtrlGeneral.bActiveStep AND (stSeqCtrlGeneral.bTimeOutActiveNoQuit OR stSeqCtrlGeneral.bTimeOutActiveQuit), 	PT:=stSeqCtrlGeneral.tTimeOut);
stSeqCtrlGeneral.tonStepTime	(IN:= stSeqCtrlGeneral.bActiveStep, PT:= T#24H);

IF stSeqCtrlGeneral.tonTimeOut.Q  THEN
	stSeqCtrlGeneral.eActiveSeqState:=E_SEQ_GENERAL.TIME_OUT;
END_IF

IF stSeqCtrlGeneral.iError<>0 THEN
	eSeq:=E_SEQ_ENGINE.ERROR_SEQ;
END_IF



eLastSeq					:=	eSeq;
stSeqCtrlGeneral.eLastActiveSeqState			:=	stSeqCtrlGeneral.eActiveSeqState;
stSeqCtrlGeneral.iLastInternalSeqStateCase	:=	stSeqCtrlGeneral.iInternalSeqStateCase;

// Reset set ready state
IF THIS^.stSeqCtrlGeneral.bExitSetReadyState THEN
  THIS^.stSeqCtrlGeneral.bExitSetReadyState := FALSE;
END_IF
END_METHOD

METHOD PRIVATE _m_TimeOut : BOOL
VAR_INPUT
	bTimeoutActiveToQuit:	BOOL;
	bTimeOutActiveNoQuit:	BOOL;
	tTimeOut:				TIME;	
END_VAR
THIS^.stSeqCtrlGeneral.bTimeOutActiveQuit:=	bTimeoutActiveToQuit;
THIS^.stSeqCtrlGeneral.bTimeOutActiveNoQuit:=	bTimeOutActiveNoQuit;
THIS^.stSeqCtrlGeneral.tTimeOut:=			tTimeOut;
_m_TimeOut:=FALSE;
IF THIS^.stSeqCtrlGeneral.tonTimeOut.Q THEN
	_m_TimeOut:=TRUE;
END_IF
END_METHOD

METHOD FB_init : BOOL
VAR_INPUT
	bInitRetains : BOOL; // if TRUE, the retain variables are initialized (warm start / cold start)
	bInCopyCode : BOOL;  // if TRUE, the instance afterwards gets moved into the copy code (online change)
  
  itfOpMode:											                        I_OP_MODE; 
  itfEventLogger:                                         I_EVENT_LOGGER;
  itfOn:                                                  I_BINARY_OUTPUT;
END_VAR
THIS^.itfOpMode := itfOpMode;
THIS^.itfEventLogger := itfEventLogger;
THIS^.itfOn := itfOn;
END_METHOD

METHOD M_Off : BOOL
M_Off := THIS^.stSeqCtrlGeneral.eActiveSeqState = E_SEQ_GENERAL.DONE;

// Assign input

// General
IF THIS^.stSeqCtrlGeneral.eActiveSeqState = E_SEQ_GENERAL.READY THEN
  THIS^.eNextSeq := E_SEQ_ENGINE.OFF;
  THIS^.stSeqCtrlGeneral.eActiveSeqState := E_SEQ_GENERAL.EXECUTE;
END_IF
END_METHOD

METHOD M_On : BOOL
M_On := THIS^.stSeqCtrlGeneral.eActiveSeqState = E_SEQ_GENERAL.DONE;

// Assign input

// General
IF THIS^.stSeqCtrlGeneral.eActiveSeqState = E_SEQ_GENERAL.READY THEN
  THIS^.eNextSeq := E_SEQ_ENGINE.ON;
  THIS^.stSeqCtrlGeneral.eActiveSeqState := E_SEQ_GENERAL.EXECUTE;
END_IF
END_METHOD

METHOD M_Reset : BOOL
VAR_INPUT
END_VAR
M_Reset := THIS^.stSeqCtrlGeneral.eActiveSeqState = E_SEQ_GENERAL.DONE;

// Assign input

// General
IF THIS^.stSeqCtrlGeneral.eActiveSeqState = E_SEQ_GENERAL.READY THEN
  THIS^.eNextSeq := E_SEQ_ENGINE.INIT;
  THIS^.stSeqCtrlGeneral.eActiveSeqState := E_SEQ_GENERAL.EXECUTE;
END_IF
END_METHOD

{warning 'Methodenimplementierung hinzufügen'}
(*=== Method: M_Run  ============================================

 @brief: Here is the global code (Timer, Event, Flange,...)*)
METHOD M_Run
END_METHOD

METHOD M_SetReady : BOOL
VAR_INPUT
END_VAR
M_SetReady := TRUE
              AND THIS^.stSeqCtrlGeneral.eActiveSeqState = E_SEQ_GENERAL.READY
              AND THIS^.eSeq = E_SEQ_ENGINE.BASE;

THIS^.stSeqCtrlGeneral.eActiveSeqState := E_SEQ_GENERAL.READY;
THIS^.eNextSeq := E_SEQ_ENGINE.BASE;
END_METHOD

{warning 'Eigenschaftenimplementierung hinzufügen'}
PROPERTY P_Busy : BOOL
GET
IF stSeqCtrlGeneral.eActiveSeqState = E_SEQ_GENERAL.READY THEN
  P_Busy := FALSE;
ELSE
  P_Busy := TRUE;
END_IF
END_GET
END_PROPERTY

{warning 'Eigenschaftenimplementierung hinzufügen'}
(*=== Property: P_Event  ============================================

 @param [set]: 	Set the Structure "ST_EVENT" from another Object
 @param [get]: 	Return the Structure "ST_EVENT", it contains the actual 
					event of the Object *)
PROPERTY P_Event : GenLib.ST_EVENT
GET
END_GET
SET
END_SET
END_PROPERTY

{warning 'Eigenschaftenimplementierung hinzufügen'}
(*=== Property: P_FullObjectPath  ============================================

 @param [set]: 	Set the Object Path (Clear String of Object)
 @param [get]: 	Return the Objectpath *)
PROPERTY P_FullObjectPath : STRING
GET
END_GET
SET
END_SET
END_PROPERTY

{warning 'Eigenschaftenimplementierung hinzufügen'}
(*=== Property: P_Global_Ack  ============================================

 @param [set]: 	Set the Bit for Ack from another Object
 @param [get]: 	Return the state of Ack Bit*)
PROPERTY P_Global_Ack : BOOL
GET
END_GET
SET
END_SET
END_PROPERTY

{warning 'Eigenschaftenimplementierung hinzufügen'}
(*=== Property: P_GlobalID  ============================================

 @param [set]: 	-
 @param [get]: 	Return the string of instance path*)
PROPERTY P_GlobalID : STRING
GET
END_GET
END_PROPERTY

{warning 'Eigenschaftenimplementierung hinzufügen'}
PROPERTY P_ReadyState : BOOL
GET
P_ReadyState := THIS^.stSeqCtrlGeneral.eActiveSeqState = E_SEQ_GENERAL.READY;
END_GET
END_PROPERTY

//{​​​​attribute 'monitoring' := 'call'}​​​​
PROPERTY P_State : BOOL
GET
P_State := THIS^.itfOn.P_State;
END_GET
END_PROPERTY

END_FUNCTION_BLOCK

// ---- MODULE/ACTOR_VALVE/VALVE/POU/FB_SHUTOFF_VALVE.TcPOU
FUNCTION_BLOCK FB_SHUTOFF_VALVE IMPLEMENTS I_ENGINE_VALVE
VAR //General
	{attribute 'instance-path'} 
  {attribute 'noinit'} 
	strInstancePath:									                      STRING;
	bInit: 												                          BOOL:=TRUE;
	strFullObjectPath: 								                      STRING;
	stEvent:											                          ST_EVENT;
	bAck:												                            BOOL;	
END_VAR
VAR   // From FB_init	
	itfOpMode:											                        I_OP_MODE; 
  itfEventLogger:                                         I_EVENT_LOGGER;
  itfOpen:                                                I_BINARY_OUTPUT;
  itfClose:                                               I_BINARY_OUTPUT;
  itfSensorOpened:                                        I_BINARY_SWITCH;
  itfSensorClosed:                                        I_BINARY_SWITCH;
  bNC:                                                    BOOL;
END_VAR                                      				
VAR	// Step chain control                				
  eSeq, eLastSeq, eNextSeq:					                      E_SEQ_ENGINE; 
                  				
  //eActiveSeqState, eLastActiveSeqState:                 E_SEQ_GENERAL;
	(*
  iInternalSeqStateCase, iLastInternalSeqStateCase:       INT:=0;       
	tonDelay, tonTimeOut, tonStepTime:						          TON;
	tDelay:													                        TIME := T#100MS;
	tTimeOut:												                        TIME := T#100MS;
	tTimeOutExt:											                      TIME := T#100MS;
	bDelayActive, bTimeOutActiveQuit, bTimeOutActiveNoQuit:	BOOL;//Timer Option
	bActiveStep, bDebugAcitve, bDebugNext:					        BOOL;//Debug Option
	i:														                          INT;
 	iError:													                        INT; //ERROR-CODE                    	                   		
	listLastSteps:											                    ARRAY[0..49] OF ST_LAST_STEPS;	
	strExtraInfo:											                      STRING; 
	eStep_Type:												                      E_STEP_STATE_TYPE; 
	bDebugModeActive:										                    BOOL;   
	bWaitForBreakpoint:										                  BOOL;
	bBreakpointActive:										                  BOOL;
	bDebugResume:											                      BOOL;   
	listBreakpoint:											                    ARRAY[0..10] OF  INT;    
*)
i:														                            INT;
stSeqCtrlGeneral:											                    ST_SEQ_CTRL_GEN;     	
END_VAR                                             		
VAR                                                 		
	bMethodeFromExtStarted:									                BOOL;
	bMethodeFromExtActive:									                BOOL;
	bMethodeFromExtDone:									                  BOOL;
	strTemp:												                        STRING;
END_VAR   
VAR
  stHMI:                                                  ST_HMI_VALVE;
  rLimit:                                                 REAL;
END_VAR                  	
VAR_TEMP                    	
	iTemp:										                              INT;
END_VAR

// Set FBs and Interfaces ready after switch internal step
IF stSeqCtrlGeneral.iInternalSeqStateCase <> stSeqCtrlGeneral.iLastInternalSeqStateCase AND NOT stSeqCtrlGeneral.bExitSetReadyState THEN
  IF TRUE
  //AND ...
  THEN
    stSeqCtrlGeneral.bExitSetReadyState := TRUE;
  ELSE
    RETURN;
  END_IF
END_IF

stSeqCtrlGeneral.strObject := F_CreateObjectName(strInstancePath);

// First method call
_m_SequenceManager();
//_m_SaveLastStep();

CASE eSeq OF 
  E_SEQ_VALVE.BASE:;
  
	E_SEQ_ENGINE.INIT: _m_Seq_INIT();
		IF TRUE
		AND (stSeqCtrlGeneral.eActiveSeqState = E_SEQ_GENERAL.DONE) 
		THEN
			eSeq := E_SEQ_ENGINE.BASE;
		END_IF
		
	E_SEQ_ENGINE.SETUP:;
  
	// Process
  E_SEQ_ENGINE.OPEN: _m_Seq_OPEN();
    IF TRUE
		AND (stSeqCtrlGeneral.eActiveSeqState = E_SEQ_GENERAL.DONE) 
		THEN
			eSeq := E_SEQ_VALVE.BASE;
		END_IF
    
  E_SEQ_ENGINE.CLOSE: _m_Seq_CLOSE();
    IF TRUE
		AND (stSeqCtrlGeneral.eActiveSeqState = E_SEQ_GENERAL.DONE) 
		THEN
			eSeq := E_SEQ_VALVE.BASE;
		END_IF

  // End
	E_SEQ_ENGINE.END:;
	E_SEQ_ENGINE.ERROR_SEQ:;	
END_CASE

strTemp:=TO_STRING(eSeq);

METHOD PRIVATE _m_DebugManager
VAR_INPUT
	iStepID: int;
END_VAR
IF TRUE
AND THIS^.stSeqCtrlGeneral.bDebugModeActive 
AND NOT THIS^.stSeqCtrlGeneral.bActiveStep
THEN


THIS^.stSeqCtrlGeneral.bBreakpointActive:=FALSE;

FOR i:=0 TO 10 DO
	
	IF TRUE
	AND iStepID=THIS^.stSeqCtrlGeneral.listBreakpoint[i] 
	AND iStepID<>0
	THEN
		EXIT;
	END_IF
END_FOR
IF (i<=10) THEN
	THIS^.stSeqCtrlGeneral.bBreakpointActive:=TRUE;
END_IF

END_IF
END_METHOD

METHOD PRIVATE _m_Delay : BOOL
VAR_INPUT
	DelayTime:	TIME;
END_VAR
THIS^.stSeqCtrlGeneral.bDelayActive:=TRUE;
THIS^.stSeqCtrlGeneral.tDelay:=DelayTime;
_m_Delay:=FALSE;
IF THIS^.stSeqCtrlGeneral.tonDelay.Q THEN
	_m_Delay:=TRUE;
END_IF
END_METHOD

METHOD PRIVATE _m_GeneralStepSetting : BOOL
VAR_INPUT
	StepType:			    	E_STEP_STATE_TYPE;
	InfoTextID:					STRING(20);
	EnableDebug:	   			BOOL;	
	
END_VAR
IF THIS^.stSeqCtrlGeneral.bActiveStep THEN
	THIS^.stSeqCtrlGeneral.eStep_Type:=StepType;
	THIS^.stSeqCtrlGeneral.strExtraInfo:= GenLib.F_RET_TXTLIST_ENTRY(strPortNr:='851',strID:='',strTxtLstName:=InfoTextID);
END_IF
END_METHOD

METHOD PRIVATE _m_SaveLastStep : BOOL
VAR_INPUT
END_VAR
VAR
	i: dint;
END_VAR
IF NOT THIS^.stSeqCtrlGeneral.bActiveStep THEN
	
	FOR i:=49 TO 1 BY -1 DO
			stSeqCtrlGeneral.listLastSteps[i].strStepName:=stSeqCtrlGeneral.listLastSteps[i-1].strStepName;
			stSeqCtrlGeneral.listLastSteps[i].tStepTime:=stSeqCtrlGeneral.listLastSteps[i-1].tStepTime;
			stSeqCtrlGeneral.listLastSteps[i].tDelayTime:=stSeqCtrlGeneral.listLastSteps[i-1].tDelayTime;
	END_FOR
	stSeqCtrlGeneral.listLastSteps[0].strStepName:=TO_STRING(THIS^.eSeq);
	stSeqCtrlGeneral.listLastSteps[1].tStepTime:=THIS^.stSeqCtrlGeneral.tonStepTime.ET;
	stSeqCtrlGeneral.listLastSteps[1].tStepTime:=THIS^.stSeqCtrlGeneral.tonDelay.ET;
ELSE
	stSeqCtrlGeneral.listLastSteps[0].tStepTime:=THIS^.stSeqCtrlGeneral.tonStepTime.ET;
	stSeqCtrlGeneral.listLastSteps[0].tDelayTime:=THIS^.stSeqCtrlGeneral.tonDelay.ET;	
END_IF
END_METHOD

METHOD _m_Seq_CLOSE : BOOL
VAR
  ActiveSeq: STRING;
END_VAR
//THIS^._m_GeneralStepSetting(StepType:=E_STEP_STATE_TYPE.INIT,
ActiveSeq := TO_STRING(THIS^.eSeq);

